( sName := 'a_bPitchExtremeFeatherSoftwareLimitSwitch', sClearName := 'Pitch system detected fine limit', sID := '4090', a := FALSE, b := FALSE, iGroup :=4, iSetDelay :=1, iResetDelay := 10, eResetMode := MANU, eBrakeProgram := B1, eAlarmProgram := 0, Enable := TRUE, iRepetitionNumber := 0 , iRepetitionPeriod := 10, Comment := 'Pitch system detected extreme feather limit', Param1 := (Set:=90, SetMin:=88, SetMax:=90,Comment:=''), Param2 := (Set:=87, SetMin:=87, SetMax:=88,Comment:='') ),
( sName := 'a_bPitchEncoder1Fault', sClearName := 'Pitch system Blade encoder 1', sID := '4091', a := FALSE, b := FALSE, iGroup :=4, iSetDelay :=1, iResetDelay := 1, eResetMode := MANU, eBrakeProgram := B20, eAlarmProgram := 0, Enable := TRUE, iRepetitionNumber := 0 , iRepetitionPeriod := 0, Comment := 'Pitch system Blade encoder 1', Param1 := (Set:=70, SetMin:=28, SetMax:=80,Comment:='Pitch Max motor current exceeded'), Param2 := (Set:=19, SetMin:=0, SetMax:=20,Comment:='') ),
( sName := 'a_bPitchLoadedEFCTest', sClearName := 'Pitch system loaded EFC Test', sID := '4092', a := FALSE, b := FALSE, iGroup :=4, iSetDelay :=1, iResetDelay := 100, eResetMode := MANU, eBrakeProgram := B99, eAlarmProgram := 0, Enable := TRUE, iRepetitionNumber := 0 , iRepetitionPeriod := 0, Comment := 'Pitch system loaded EFC Test', Param1 := (Set:=0, SetMin:=0, SetMax:=0,Comment:=''), Param2 := (Set:=0, SetMin:=0, SetMax:=0,Comment:='') ),
( sName := 'a_bYawDummyAlarm', sClearName := 'Water level below slip ring tripped low sensor', sID := '5001', a := FALSE, b := FALSE, iGroup :=5, iSetDelay :=50, iResetDelay := 0, eResetMode := MANU, eBrakeProgram := B99, eAlarmProgram := 0, Enable := FALSE, iRepetitionNumber := 0 , iRepetitionPeriod := 0, Comment := 'Water level below slip ring tripped low sensor at bottom of trough', Param1 := (Set:=0, SetMin:=0, SetMax:=0,Comment:=''), Param2 := (Set:=0, SetMin:=0, SetMax:=0,Comment:='') ),
( sName := 'a_bLSSDummyAlarm', sClearName := '', sID := '6002', a := FALSE, b := FALSE, iGroup :=5, iSetDelay :=50, iResetDelay := 0, eResetMode := MANU, eBrakeProgram := B100, eAlarmProgram := EMAIL, Enable := FALSE, iRepetitionNumber := 0 , iRepetitionPeriod := 0, Comment := 'Ambient temperature high at front of nacelle', Param1 := (Set:=40, SetMin:=0, SetMax:=100,Comment:=''), Param2 := (Set:=0, SetMin:=0, SetMax:=0,Comment:='') ),
( sName := 'a_bGENDummyAlarm', sClearName := '', sID := '15001', a := FALSE, b := FALSE, iGroup :=5, iSetDelay :=50, iResetDelay := 0, eResetMode := MANU, eBrakeProgram := B100, eAlarmProgram := EMAIL, Enable := FALSE, iRepetitionNumber := 0 , iRepetitionPeriod := 0, Comment := 'Ambient temperature high at front of nacelle', Param1 := (Set:=40, SetMin:=0, SetMax:=100,Comment:=''), Param2 := (Set:=0, SetMin:=0, SetMax:=0,Comment:='') ),
( sName := 'a_bGearDummyAlarm', sClearName := '', sID := '8001', a := FALSE, b := FALSE, iGroup :=5, iSetDelay :=50, iResetDelay := 0, eResetMode := MANU, eBrakeProgram := B100, eAlarmProgram := EMAIL, Enable := FALSE, iRepetitionNumber := 0 , iRepetitionPeriod := 0, Comment := 'Ambient temperature high at front of nacelle', Param1 := (Set:=40, SetMin:=0, SetMax:=100,Comment:=''), Param2 := (Set:=0, SetMin:=0, SetMax:=0,Comment:='') ),
( sName := 'a_bAuxPowerBreakerError_2S1_MainSwitch', sClearName := '2S1', sID := '9001', a := FALSE, b := FALSE, iGroup :=9, iSetDelay :=0, iResetDelay := 0, eResetMode := MANU, eBrakeProgram := B99, eAlarmProgram := 0, Enable := TRUE, iRepetitionNumber := 0 , iRepetitionPeriod := 10, Comment := 'Main Supply Switch', Param1 := (Set:=0, SetMin:=0, SetMax:=0,Comment:=''), Param2 := (Set:=0, SetMin:=0, SetMax:=0,Comment:='') ),
( sName := 'a_bAuxPowerDCbusSupply01Fault', sClearName := 'a_bAuxPowerPriDCbusSupply01Fault', sID := '9038', a := FALSE, b := FALSE, iGroup :=9, iSetDelay :=30, iResetDelay := 0, eResetMode := MANU, eBrakeProgram := B99, eAlarmProgram := 0, Enable := TRUE, iRepetitionNumber := 0 , iRepetitionPeriod := 10, Comment := '', Param1 := (Set:=0, SetMin:=0, SetMax:=0,Comment:=''), Param2 := (Set:=0, SetMin:=0, SetMax:=0,Comment:='') ),
( sName := 'a_bAuxPowerDCbusUPS1AlarmActive', sClearName := 'a_bAuxPowerPriDCbusUPS1AlarmActive', sID := '9039', a := FALSE, b := FALSE, iGroup :=9, iSetDelay :=0, iResetDelay := 0, eResetMode := MANU, eBrakeProgram := B99, eAlarmProgram := 0, Enable := TRUE, iRepetitionNumber := 0 , iRepetitionPeriod := 10, Comment := '', Param1 := (Set:=0, SetMin:=0, SetMax:=0,Comment:=''), Param2 := (Set:=0, SetMin:=0, SetMax:=0,Comment:='') ),
( sName := 'a_bAuxPowerDCbusUPS1BatteryLow', sClearName := 'a_bAuxPowerPriDCbusUPS1BatteryLow', sID := '9040', a := FALSE, b := FALSE, iGroup :=9, iSetDelay :=30, iResetDelay := 0, eResetMode := MANU, eBrakeProgram := B99, eAlarmProgram := 0, Enable := TRUE, iRepetitionNumber := 0 , iRepetitionPeriod := 10, Comment := '', Param1 := (Set:=0, SetMin:=0, SetMax:=0,Comment:=''), Param2 := (Set:=0, SetMin:=0, SetMax:=0,Comment:='') ),
( sName := 'a_bAuxPowerDCbusUPS1BatteryLifeWarning', sClearName := 'a_bAuxPowerPriDCbusUPS1BatteryLifeWarning', sID := '9041', a := FALSE, b := FALSE, iGroup :=9, iSetDelay :=0, iResetDelay := 0, eResetMode := MANU, eBrakeProgram := B99, eAlarmProgram := 0, Enable := TRUE, iRepetitionNumber := 0 , iRepetitionPeriod := 10, Comment := '', Param1 := (Set:=0, SetMin:=0, SetMax:=0,Comment:=''), Param2 := (Set:=0, SetMin:=0, SetMax:=0,Comment:='') ),
( sName := 'a_bAuxPowerDCbusUPS1BatteryLifeLoLo', sClearName := 'a_bAuxPowerPriDCbusUPS1BatteryLifeLoLo', sID := '9042', a := FALSE, b := FALSE, iGroup :=9, iSetDelay :=0, iResetDelay := 0, eResetMode := MANU, eBrakeProgram := B99, eAlarmProgram := 0, Enable := TRUE, iRepetitionNumber := 0 , iRepetitionPeriod := 10, Comment := '', Param1 := (Set:=0, SetMin:=0, SetMax:=0,Comment:=''), Param2 := (Set:=0, SetMin:=0, SetMax:=0,Comment:='') ),
( sName := 'a_bAuxPowerDCbusUPS1BatteryCharging', sClearName := 'a_bAuxPowerPriDCbusUPS1BatteryCharging', sID := '9043', a := FALSE, b := FALSE, iGroup :=9, iSetDelay :=100, iResetDelay := 0, eResetMode := MANU, eBrakeProgram := B99, eAlarmProgram := 0, Enable := TRUE, iRepetitionNumber := 0 , iRepetitionPeriod := 10, Comment := '', Param1 := (Set:=0, SetMin:=0, SetMax:=0,Comment:=''), Param2 := (Set:=0, SetMin:=0, SetMax:=0,Comment:='') ),
( sName := 'a_bAuxPowerDCbusUPS1BatteryChargingTooLong', sClearName := 'a_bAuxPowerPriDCbusUPS1BatteryChargingTooLong', sID := '9044', a := FALSE, b := FALSE, iGroup :=9, iSetDelay :=108000, iResetDelay := 0, eResetMode := MANU, eBrakeProgram := B99, eAlarmProgram := 0, Enable := TRUE, iRepetitionNumber := 0 , iRepetitionPeriod := 10, Comment := '', Param1 := (Set:=0, SetMin:=0, SetMax:=0,Comment:=''), Param2 := (Set:=0, SetMin:=0, SetMax:=0,Comment:='') ),
( sName := 'a_bAuxPowerDCbusORing01RedunFault', sClearName := 'a_bAuxPowerPriDCbusORing01RedunFault', sID := '9045', a := FALSE, b := FALSE, iGroup :=9, iSetDelay :=0, iResetDelay := 0, eResetMode := MANU, eBrakeProgram := B99, eAlarmProgram := 0, Enable := TRUE, iRepetitionNumber := 0 , iRepetitionPeriod := 10, Comment := '', Param1 := (Set:=0, SetMin:=0, SetMax:=0,Comment:=''), Param2 := (Set:=0, SetMin:=0, SetMax:=0,Comment:='') ),
( sName := 'a_bAuxPowerDCbusORing01RedunWarning', sClearName := 'a_bAuxPowerPriDCbusORing01RedunWarning', sID := '9046', a := FALSE, b := FALSE, iGroup :=9, iSetDelay :=0, iResetDelay := 0, eResetMode := MANU, eBrakeProgram := B99, eAlarmProgram := 0, Enable := TRUE, iRepetitionNumber := 0 , iRepetitionPeriod := 10, Comment := '', Param1 := (Set:=0, SetMin:=0, SetMax:=0,Comment:=''), Param2 := (Set:=0, SetMin:=0, SetMax:=0,Comment:='') ),
( sName := 'a_bAuxPowerDCbusDCVoltageLow', sClearName := '', sID := '9074', a := FALSE, b := FALSE, iGroup :=9, iSetDelay :=0, iResetDelay := 0, eResetMode := MANU, eBrakeProgram := B99, eAlarmProgram := 0, Enable := TRUE, iRepetitionNumber := 0 , iRepetitionPeriod := 10, Comment := '24VDC Bus Low Voltage Detected', Param1 := (Set:=23, SetMin:=22, SetMax:=30,Comment:='DC Bus Voltage Low'), Param2 := (Set:=0, SetMin:=0, SetMax:=0,Comment:='') ),
( sName := 'a_bStatusBackupChargerAxis1CriticalError', sClearName := 'a_bStatusBackupChargerAxis1CriticalError', sID := '9074', a := FALSE, b := FALSE, iGroup :=9, iSetDelay :=0, iResetDelay := 0, eResetMode := MANU, eBrakeProgram := B1, eAlarmProgram := 0, Enable := TRUE, iRepetitionNumber := 0 , iRepetitionPeriod := 10, Comment := 'a_bStatusBackupChargerAxis1CriticalError', Param1 := (Set:=0, SetMin:=0, SetMax:=0,Comment:=''), Param2 := (Set:=0, SetMin:=0, SetMax:=0,Comment:='') ),
( sName := 'a_bGridLossDetected', sClearName := '', sID := '10001', a := FALSE, b := FALSE, iGroup :=10, iSetDelay :=0, iResetDelay := 0, eResetMode := MANU, eBrakeProgram := B17, eAlarmProgram := 0, Enable := TRUE, iRepetitionNumber := 0 , iRepetitionPeriod := 10, Comment := 'Grid loss detected by converter', Param1 := (Set:=0, SetMin:=0, SetMax:=0,Comment:=''), Param2 := (Set:=0, SetMin:=0, SetMax:=0,Comment:='') ),
( sName := 'a_bLowVoltageRideThrough', sClearName := '', sID := '10002', a := FALSE, b := FALSE, iGroup :=10, iSetDelay :=0, iResetDelay := 0, eResetMode := MANU, eBrakeProgram := B99, eAlarmProgram := 0, Enable := TRUE, iRepetitionNumber := 0 , iRepetitionPeriod := 10, Comment := 'LVRT detected by converter', Param1 := (Set:=0, SetMin:=0, SetMax:=0,Comment:=''), Param2 := (Set:=0, SetMin:=0, SetMax:=0,Comment:='') ),
( sName := 'a_bScadaEnableAutoStartRequested', sClearName := '', sID := '11001', a := FALSE, b := FALSE, iGroup :=11, iSetDelay :=0, iResetDelay := 0, eResetMode := MANU, eBrakeProgram := B99, eAlarmProgram := 0, Enable := TRUE, iRepetitionNumber := 0 , iRepetitionPeriod := 0, Comment := 'SCADA enable autostart requested', Param1 := (Set:=0, SetMin:=0, SetMax:=0,Comment:=''), Param2 := (Set:=0, SetMin:=0, SetMax:=0,Comment:='') ),
( sName := 'a_bScadaDisableAutoStartRequested', sClearName := '', sID := '11002', a := FALSE, b := FALSE, iGroup :=11, iSetDelay :=0, iResetDelay := 0, eResetMode := MANU, eBrakeProgram := B99, eAlarmProgram := 0, Enable := TRUE, iRepetitionNumber := 0 , iRepetitionPeriod := 0, Comment := 'SCADA disable autostart requested', Param1 := (Set:=0, SetMin:=0, SetMax:=0,Comment:=''), Param2 := (Set:=0, SetMin:=0, SetMax:=0,Comment:='') ),
( sName := 'a_bScadaNormalStopRequested', sClearName := '', sID := '11003', a := FALSE, b := FALSE, iGroup :=11, iSetDelay :=0, iResetDelay := 0, eResetMode := MANU, eBrakeProgram := B99, eAlarmProgram := 0, Enable := TRUE, iRepetitionNumber := 0 , iRepetitionPeriod := 0, Comment := 'SCADA normal stop requested', Param1 := (Set:=0, SetMin:=0, SetMax:=0,Comment:=''), Param2 := (Set:=0, SetMin:=0, SetMax:=0,Comment:='') ),
( sName := 'a_bScadaAlarmResetRequested', sClearName := '', sID := '11004', a := FALSE, b := FALSE, iGroup :=11, iSetDelay :=0, iResetDelay := 0, eResetMode := MANU, eBrakeProgram := B99, eAlarmProgram := 0, Enable := TRUE, iRepetitionNumber := 0 , iRepetitionPeriod := 0, Comment := 'SCADA alarm reset requested', Param1 := (Set:=0, SetMin:=0, SetMax:=0,Comment:=''), Param2 := (Set:=0, SetMin:=0, SetMax:=0,Comment:='') ),
( sName := 'a_bScadaSafetyResetRequested', sClearName := '', sID := '11005', a := FALSE, b := FALSE, iGroup :=11, iSetDelay :=0, iResetDelay := 0, eResetMode := MANU, eBrakeProgram := B99, eAlarmProgram := 0, Enable := TRUE, iRepetitionNumber := 0 , iRepetitionPeriod := 0, Comment := 'SCADA safety reset requested', Param1 := (Set:=0, SetMin:=0, SetMax:=0,Comment:=''), Param2 := (Set:=0, SetMin:=0, SetMax:=0,Comment:='') ),
( sName := 'a_bScadaOpModeChangeRequested', sClearName := '', sID := '11006', a := FALSE, b := FALSE, iGroup :=11, iSetDelay :=0, iResetDelay := 0, eResetMode := MANU, eBrakeProgram := B99, eAlarmProgram := 0, Enable := TRUE, iRepetitionNumber := 0 , iRepetitionPeriod := 0, Comment := 'SCADA op mode change requested', Param1 := (Set:=0, SetMin:=0, SetMax:=0,Comment:=''), Param2 := (Set:=0, SetMin:=0, SetMax:=0,Comment:='') ),
( sName := 'a_bScadaServiceIdleStRequest', sClearName := '', sID := '11007', a := FALSE, b := FALSE, iGroup :=11, iSetDelay :=0, iResetDelay := 0, eResetMode := MANU, eBrakeProgram := B99, eAlarmProgram := 0, Enable := TRUE, iRepetitionNumber := 0 , iRepetitionPeriod := 0, Comment := 'SCADA service idle ST request', Param1 := (Set:=0, SetMin:=0, SetMax:=0,Comment:=''), Param2 := (Set:=0, SetMin:=0, SetMax:=0,Comment:='') ),
( sName := 'a_bScadaServiceStopStRequest', sClearName := '', sID := '11008', a := FALSE, b := FALSE, iGroup :=11, iSetDelay :=0, iResetDelay := 0, eResetMode := MANU, eBrakeProgram := B99, eAlarmProgram := 0, Enable := TRUE, iRepetitionNumber := 0 , iRepetitionPeriod := 0, Comment := 'SCADA service stop ST request', Param1 := (Set:=0, SetMin:=0, SetMax:=0,Comment:=''), Param2 := (Set:=0, SetMin:=0, SetMax:=0,Comment:='') ),
( sName := 'a_bScadaEnableSafetyNACPRequested', sClearName := '', sID := '11009', a := FALSE, b := FALSE, iGroup :=11, iSetDelay :=0, iResetDelay := 0, eResetMode := MANU, eBrakeProgram := B99, eAlarmProgram := 0, Enable := TRUE, iRepetitionNumber := 0 , iRepetitionPeriod := 0, Comment := 'SCADA enable safety NACP requested', Param1 := (Set:=0, SetMin:=0, SetMax:=0,Comment:=''), Param2 := (Set:=0, SetMin:=0, SetMax:=0,Comment:='') ),
( sName := 'a_bScadaDisableSafetyNACPRequested', sClearName := '', sID := '11010', a := FALSE, b := FALSE, iGroup :=11, iSetDelay :=0, iResetDelay := 0, eResetMode := MANU, eBrakeProgram := B99, eAlarmProgram := 0, Enable := TRUE, iRepetitionNumber := 0 , iRepetitionPeriod := 0, Comment := 'SCADA disable safety NACP requested', Param1 := (Set:=0, SetMin:=0, SetMax:=0,Comment:=''), Param2 := (Set:=0, SetMin:=0, SetMax:=0,Comment:='') ),
( sName := 'a_bScadaEnableSafetyNACSRequested', sClearName := '', sID := '11011', a := FALSE, b := FALSE, iGroup :=11, iSetDelay :=0, iResetDelay := 0, eResetMode := MANU, eBrakeProgram := B99, eAlarmProgram := 0, Enable := TRUE, iRepetitionNumber := 0 , iRepetitionPeriod := 0, Comment := 'SCADA enable safety NACS requested', Param1 := (Set:=0, SetMin:=0, SetMax:=0,Comment:=''), Param2 := (Set:=0, SetMin:=0, SetMax:=0,Comment:='') ),
( sName := 'a_bScadaDisableSafetyNACSRequested', sClearName := '', sID := '11012', a := FALSE, b := FALSE, iGroup :=11, iSetDelay :=0, iResetDelay := 0, eResetMode := MANU, eBrakeProgram := B99, eAlarmProgram := 0, Enable := TRUE, iRepetitionNumber := 0 , iRepetitionPeriod := 0, Comment := 'SCADA disable safety NACS requested', Param1 := (Set:=0, SetMin:=0, SetMax:=0,Comment:=''), Param2 := (Set:=0, SetMin:=0, SetMax:=0,Comment:='') ),
( sName := 'a_bScadaLossOfCommsToTTGC', sClearName := '', sID := '11013', a := FALSE, b := FALSE, iGroup :=11, iSetDelay :=0, iResetDelay := 0, eResetMode := MANU, eBrakeProgram := B99, eAlarmProgram := 0, Enable := TRUE, iRepetitionNumber := 0 , iRepetitionPeriod := 0, Comment := 'SCADA loss of comms to TTGC', Param1 := (Set:=0, SetMin:=0, SetMax:=0,Comment:=''), Param2 := (Set:=0, SetMin:=0, SetMax:=0,Comment:='') )];
iMaxAlarms: INT := 222;
arrAlarmStatus: ARRAY [1..222] OF BOOL;
arrAlarmGroup: ARRAY [1..222] OF INT;
END_VAR

// ---- Alarm System/GVLs/A. Operation/01_General/GlobVar_GeneralLog_Privat.TcGVL
{attribute 'Tc2GvlVarNames'}
VAR_GLOBAL	(*GlobVar_GeneralLog_Privat*)

(*-------------  General  / multiple variables  for Operation  --------------------------------------------------------*)

	Lib_rGeneratorPower: 		REAL;
	Lib_rGeneratorSpeed: 		REAL;
	Lib_rFlowSpeed: 			REAL;
(*	Lib_rPitchAngle: 			REAL;	*)


(*-------------  General Log variables  --------------------------------------------------------------------------------------*)

	(* Turbine Identification (Header for log  files):	*)
	Lib_st_xTurbineIdent : 			ST_xTurbineIdent;

	(* System Time:   ---------------------------------------------*)
	Lib_strucSystemTime: 		TIMESTRUCT;
	Lib_sOffsetUTC:			STRING[20];
	Lib_sLocalTime: 			STRING[24];
	Lib_sTimeZoneInfo:		STRING[20];

	(* Operating System:   --------------------------------------*)
	Lib_OperatingSystemCEDetected: 	BOOL;		(*NSM 231016*)
	g_dtLocalTime :DT;
	g_iLocalTime: UDINT;
	g_fLocalTime: LREAL;

(*-------------   In General need for all Logger  --------------------------------------------------------------------------------*)

	LibDetectNewYear	:	BOOL;
	LibDetectNewMonth	:	BOOL;
	LibDetectNewDay		:	BOOL;
	LibDetectNewHour	:	BOOL;
	LibDetectNew10min	:	BOOL;
	LibDetectNew5min	:	BOOL;
	LibDetectNewMinute	:	BOOL;
	LibDetectNew30sec	:	BOOL;
	LibDetectNewSecond	:	BOOL;
	LibDetectNew100ms	:	BOOL;

(* --------------------------------------------------------------------------------------------------------------------------------------*)

END_VAR

// ---- Alarm System/GVLs/A. Operation/01_General/GlobVar_LibStatuscodeLogger_Privat.TcGVL
{attribute 'Tc2GvlVarNames'}
VAR_GLOBAL CONSTANT	(*GlobVar_LibPowerCurves_Privat*)

	guiKeyAndTextLen					: UINT := 91; 		(*max using length for Statuscode description is [uiKeyAndTextLen - sKeySize, e.g. 001-005-280]*)
	NUMBER_OF_EVENT_DATAS			: UINT := 4; 		(* number of process values  *)
	giGeneralLoggerChannelInUsed			: UINT := 75; 		(* how many  channels  the log file max. can contain*)
(*	giNumberOfStatuscodes				: UINT := 850;		*)

	giCountsOfKeyLetterForStatuscodeFile 	: UINT := 75; 		(* Length of minimize Key-string in the file better reading in the text file *)
	giSizeARRListOfStatuscodesToBeSent: 	USINT:= 50;		(*must be tuned to the number given for the ARRAY*)
	guiStrBufferSize: 						UINT:= 47000;		(*length of buffer for statuscode file writing *) (* header 1100 + row 200 * 218 sign = 44700*)

	giHeaderLineLenght					: UINT := 100;		(*length of each line in the header, not the column description*)
	giHeaderColumnLineLEN				: UINT :=4096; 	(*length of column text in the header *)
	giGeneralLenghtOfName				: UINT := 40; 		(* lenght of the column description name *)

END_VAR
VAR_GLOBAL PERSISTENT
//	gxStatuscode		: 				ARRAY[1..850] OF STRUC_Statuscode;
	arrAllListsOfStatuscodesToBeSent: 	ARRAY [1..3] OF ARR_ListOfStatuscodesToBeSent;	(*List of triggered Statuscodes to be sent*)
END_VAR
VAR_GLOBAL

(*  Statuscode Logger:	*)
	gsSC_PathName						: T_MaxString ;	(* Set the Path name in the init program *)
(*	gsSCunlimited_PathName 				: T_MaxString ;	(* Set the Path name with the actual day in the name *)
	gsSCunlimited_PathNameEmbeddedPC	: T_MaxString		:= '\Hard Disk\WEC_Data\Statuscode\';
	gsSCunlimited_PathNamePC 			: T_MaxString 	:='C:\temp\WEC_Data\Statuscode\'; (*Set general name without extension; .txt*)
*)

(*  General Set Values:	*)
	CheckMemCpy_Min	: UDINT;
	CheckMemCpy_Max	: UDINT;
	iOneEntrySize		: INT;
	iOneEntryLength		: INT;

	fbSCLogger					: FB_StatusCodeLogger;
	gwNewDayForLogger    		: WORD; 			(*For detection if we have a new day*)
	giRingBufferFileOneEntryLength 	: UINT; 			(*Length of one entry in the ring buffer Statuscode file*)
	giRingBufferFileHeaderLEN		: INT; 			(*Length of the whole header = header description + column description*)

//	arLoggedSC	 : 				ARRAY[1..400] OF ST_LoggedEvent_SC;	(* Logged Trigger Event *)(* twice(200) - Normal and Transfer Buffers *)
	gstrRingBufferFileColumnText: 	T_MaxString; 		(*first part of column decription*)



	giPointer1AlarmList1: USINT;
	giPointer2AlarmList1: USINT;
	giPointer3AlarmList1: USINT;
	giPointer4AlarmList1: USINT;
	giPointer5AlarmList1: USINT;
	giPointer6AlarmList1: USINT;
	giPointer7AlarmList1: USINT;
	giPointer8AlarmList1: USINT;
	giPointer9AlarmList1: USINT;
	giPointer10AlarmList1: USINT;

	giPointer1AlarmList2: USINT;
	giPointer2AlarmList2: USINT;
	giPointer3AlarmList2: USINT;
	giPointer4AlarmList2: USINT;
	giPointer5AlarmList2: USINT;
	giPointer6AlarmList2: USINT;
	giPointer7AlarmList2: USINT;
	giPointer8AlarmList2: USINT;
	giPointer9AlarmList2: USINT;
	giPointer10AlarmList2: USINT;

	giPointer1AlarmList3: USINT;
	giPointer2AlarmList3: USINT;
	giPointer3AlarmList3: USINT;
	giPointer4AlarmList3: USINT;
	giPointer5AlarmList3: USINT;
	giPointer6AlarmList3: USINT;
	giPointer7AlarmList3: USINT;
	giPointer8AlarmList3: USINT;
	giPointer9AlarmList3: USINT;
	giPointer10AlarmList3: USINT;

	giPointer_fbSendAlarmBuffer1:		USINT;		(*TO_BE_DONE__HP*)	(*pointer must be managed ?????*)
	giPointer_fbSendAlarmBuffer2:		USINT;								(*pointer must be managed ? ? ? ? ?*)
	giPointer_fbSendAlarmBuffer3:		USINT;								(*pointer must be managed ? ? ? ? ?*)


END_VAR

// ---- Alarm System/GVLs/A. Operation/01_General/GVL_Static.TcGVL
{attribute 'Tc2GvlVarNames'}
VAR_GLOBAL
	g_btempAlarmTrig:BOOL;
END_VAR

// ---- Alarm System/GVLs/A. Operation/01_General/ProgramVersions.TcGVL
{attribute 'Tc2GvlVarNames'}
VAR_GLOBAL PERSISTENT

	arrProgramVersions: ARRAY [1..20] OF ST_ProgramVersions :=[
(sVersionDate := '2021_04_21', sChangesMade := '')];
	iMaxProgVersions: INT := 20;
END_VAR

// ---- Alarm System/GVLs/A. Operation/01_General/TurbineData.TcGVL
{attribute 'Tc2GvlVarNames'}
(*VAR_GLOBAL PERSISTENT
 {attribute 'OPC.UA.DA' := '1'}
	stTurbineData: ST_TurbineData :=
	(sOperAlarmParkName :='',
	sOperAlarmTurbineName :='',
	sOperAlarmParkId :='',
	sOperAlarmTurbineId :='',
	sOperCountryCode :='',
	sOperTurbineManufacturer :='',
	sOperTurbineType :='',
	sOperBladeType := '',
	sOperInverterType := '',
	sOperTowerType := '',
	sOperTowerBearing := '',
	sTower1stBendFreg := '',
	sTower2ndBendFreg := '',
	sPitchGenNomSpeed := '');		

END_VAR
*)

VAR_GLOBAL
//	g_stTurbineRelatedData: ST_TurbineRelatedData;
 {attribute 'OPC.UA.DA' := '1'}
	g_bOperTurbineCommsFault: BOOL;
	 {attribute 'OPC.UA.DA' := '1'}
	g_fOperTurbineCapacityFactor :REAL;
   {attribute 'OPC.UA.DA' := '1'}
	g_fOperTurbineTotalEnergyGenerated :REAL;
   {attribute 'OPC.UA.DA' := '1'}
	g_tOperTurbineTimeSpentInFaultState :TIME;
   {attribute 'OPC.UA.DA' := '1'}
	g_tOperTurbineTimeSpentInOffState :TIME;
   {attribute 'OPC.UA.DA' := '1'}
	g_tOperTurbineTimeSpentInProduction :TIME;  

END_VAR

// ---- Alarm System/GVLs/GVL_EventLogger.TcGVL
{attribute 'qualified_only'}
VAR_GLOBAL
	cMaxNumberOfEvent:UINT; //
	
	
	
END_VAR

// ---- Base/Example/GVL/GVL_HMI.TcGVL
{attribute 'qualified_only'}
VAR_GLOBAL
	(*IO*)
	stTest04_DigitalInput:stHMI_DigitalInput;
	stTest05_DigitalInput:stHMI_DigitalInput;
	
	(*SYSTEM*)
	stTest01_Intlk:stHMI_Interlock;
	stTest02_Perm:stHMI_Permissive;
	stTest03_RunCtrl:stHMI_SystemRunControl;
END_VAR

// ---- MAIN.TcPOU
PROGRAM MAIN
VAR
	
END_VAR

POU_TestBase();

//AlarmWithCustomSourceInfo();
//OtherAlarmsWithCustomSource();
P_AlarmHandling();
P_AlarmTable();
MultipleAlarmCreation();

P_EventLogger_TCSAlarms();

END_PROGRAM

// ---- Base/Example/POU/POU_TestBase.TcPOU
PROGRAM POU_TestBase
VAR
	fbTestAI:fbIO_AnalogueInput;
	fbTestIntlk:FB_Interlock;	
	fbTestPerm:FB_Permissive;
	fbTestRunCtrl:FB_SystemRunControl;
	fbTestDigitalInput:fbIO_DigitalInput;
	HMI_AI_001:stHMI_AnalogueInput;
	ERROR_AI_001:stError_AnalogueInput;
	fbTestAO:fbIO_AnalogueOutput;
	HMI_DI_001:stHMI_DigitalInput;
	pulseTest:fbPulser;
	HMI_DO_001:stHMI_DigitalOutput;
	fbTestDO:fbIO_DigitalOutput;
	testAlarmset:FB_AlarmEventSet;
	bHMITest:BOOL;
	bPLCTest:BOOL;
	
	test_Valve:fbValve_Solenoid;
	HMI_XV_001:stHMI_ValveControl;
	Error_XV_001:stError_Valve;
END_VAR

testAlarmset(bAlarmEventTrigger:= , tSetDelay:= , tResetDelay:= , bOutAlarmEvent=> );

test_Valve(
	tInTimeout:= , 
	iInMode:= , 
	bInEstop:= , 
	bInSignalHome:= , 
	bInSignalWork:= , 
	bInEnable:= , 
	bInCommandWork:= , 
	bInResetError:= , 
	bInSimulate:= , 
	bOutCommandHome=> , 
	bOutCommandWork=> , 
	bOutActiveHome=> , 
	bOutActiveWork=> , 
	bOutAuto=> , 
	bOutError=> , 
	ERROR_Valve=>Error_XV_001 , 
	HMI_ValveControl:=HMI_XV_001 );

fbTestDigitalInput(
	iInMode:= , 
	bInInput:= , 
	tInOnDebounce:= , 
	tInOffDebounce:= , 
	bOutAuto=> , 
	bOutOn=> , 
	bOutRisingEdge=> , 
	bOutFallingEdge=> , 
	HMI_DigitalInput:=HMI_DI_001 );

fbTestAI(
	iInMode:= , 
	iInValue:= , 
	iInSensorType:= , 
	rInEngUnitsMin:= , 
	rInEngUnitsMax:= , 
	rInLowLow:= , 
	rInLow:= , 
	rInHigh:= , 
	rInHighHigh:= , 
	rInLowLowDeadband:= , 
	rInLowDeadband:= , 
	rInHighDeadband:= , 
	rInHighHighDeadband:= , 
	bInResetError:= , 
	rOutEngUnitsValue=> , 
	bOutLowLow=> , 
	bOutLow=> , 
	bOutHigh=> , 
	bOutHighHigh=> , 
	bOutAuto=> , 
	bOutError=> , 
	ERROR_IO_AnalogueIn=>ERROR_AI_001 , 
	HMI_IO_AnalogueInput:=HMI_AI_001 );
	
fbTestIntlk(
	bInterlock1:= , 
	bInterlock2:= , 
	bInterlock3:= , 
	bInterlock4:= , 
	bInterlock5:= , 
	bInterlock6:= , 
	bInterlock7:= , 
	bInterlock8:= , 
	bInterlock9:= , 
	bInterlock10:= , 
	bInterlock11:= , 
	bInterlock12:= , 
	bInterlock13:= , 
	bInterlock14:= , 
	bInterlock15:= , 
	bInterlock16:= , 
	bOutInterlockOk=> , 
	HMI_Interlock:=GVL_HMI.stTest01_Intlk );

fbTestPerm(
	bPermissive1:= , 
	bPermissive2:= , 
	bPermissive3:= , 
	bPermissive4:= , 
	bPermissive5:= , 
	bPermissive6:= , 
	bPermissive7:= , 
	bPermissive8:= , 
	bPermissive9:= , 
	bPermissive10:= , 
	bPermissive11:= , 
	bPermissive12:= , 
	bPermissive13:= , 
	bPermissive14:= , 
	bPermissive15:= , 
	bPermissive16:= , 
	bOutPermissiveOk=>, 
	HMI_Permissive:= GVL_HMI.stTest02_Perm);

GVL_HMI.stTest01_Intlk.asInterlockNames[1]:='Valve in correct pos';
	
fbTestRunCtrl(
	bInEnableStart:= , 
	bInEnableStop:= , 
	bInStartAuto:= , 
	bInStopAuto:= , 
	bOutRunCmd=> , 
	HMI_SystemRunControl:= GVL_HMI.stTest03_RunCtrl);
	
fbTestDO(
	iInMode:= , 
	bInEstop:= , 
	bInEnable:= , 
	bInCommand:= , 
	bOutAuto=> , 
	bOutCommand=> , 
	HMI_IO_DigitalOutput:=HMI_DO_001 );

pulseTest(
	bInRun:= , 
	tInTimeOn:=T#5S , 
	tInTimeOff:=T#10S , 
	iInNumPulses:= , 
	bOutPulse=> , 
	bOutDone=> , 
	iOutCount=> );
	
	POu();

END_PROGRAM

// ---- Base/IO/POU/fbIO_AnalogueInput.TcPOU
FUNCTION_BLOCK fbIO_AnalogueInput
VAR_INPUT
	iInMode:		INT;
	iInValue:		INT;
	iInSensorType:	INT;
	rInEngUnitsMin:	REAL;
	rInEngUnitsMax:	REAL;
	rInLowLow:		REAL;
	rInLow:			REAL;
	rInHigh:		REAL;
	rInHighHigh:	REAL;
	rInLowLowDeadband: REAL;
	rInLowDeadband:REAL;
	rInHighDeadband:REAL;
	rInHighHighDeadband:REAL;
	bInResetError:BOOL;
END_VAR
VAR_OUTPUT
	rOutEngUnitsValue:REAL; (*Engineering units scaled value*)
	bOutLowLow:BOOL; (*Low low alarm is active*)
	bOutLow:BOOL; (*Low warning is active*)
	bOutHigh:BOOL; (*High warning is active*)
	bOutHighHigh:BOOL; (*High high alarm is active*)
	bOutAuto:BOOL; (*Input is in auto mode*)
	bOutError:BOOL; (*Error Exists*)
	ERROR_IO_AnalogueIn:stError_AnalogueInput;
END_VAR

VAR_IN_OUT
	HMI_IO_AnalogueInput:stHMI_AnalogueInput;
END_VAR

VAR
	fScaled16:REAL;
	fTempScaled16:REAL;
	ftempScaled16_a:REAL;
	ftempScaled16_b:REAL;
	bTest:BOOL;
END_VAR

//Process Alarms limits
bOutLowLow:= (rOutEngUnitsValue<=(rInLowLow-rInLowLowDeadband));  	// LL Alarm
bOutLow:= (rOutEngUnitsValue<=(rInLow-rInLowDeadband));  			// LL Warning
bOutHighHigh:= (rOutEngUnitsValue>=(rInHigh+rInHighHighDeadband));  	// HH Alarm	
bOutHigh:= (rOutEngUnitsValue>=(rInHighHigh+rInHighDeadband));  		// HH Warning	
	
bOutAuto := iInMode=1;

(***************************SCALING ANALOGUE************************
ftempScaled16_a:=
ftempScaled16_b:=
IF fTempScaled32 THEN
	
END_IF
*)
(*
CASE iInMode OF
	0:
		;
	1:	// Auto mode
		rOutEngUnitsValue:=fScaled16;
	2:	// Manual Mode
		rOutEngUnitsValue:=HMI_IO_AnalogueInput.rManualValue;
		
	3:	// Independant
	END_CASE
*)

(*control bOut based on the global input and HMI input mode*)
(*if in independant mode allow control of the output based on HMI commands (MANUAL) AND digital input (AUTO)*)
IF iInMode=10 THEN
	//if HMI requests manual mode 
	IF HMI_IO_AnalogueInput.iMode=2 THEN
		;
	ELSE
		;
	END_IF
ELSE
	//bOutOn:=tonInOnDebounce.Q OR tofInOnDebounce.Q;
END_IF
	


(*Map Error bits*)
ERROR_IO_AnalogueIn.LowLowAlarm:=bOutLowLow;			//HH alarm
ERROR_IO_AnalogueIn.HighHighAlarm:=bOutHighHigh;		//LL Alarm	
	
(*map active value to the scada*)
HMI_IO_AnalogueInput.rInputValue:=fScaled16;
HMI_IO_AnalogueInput.rActiveValue:=rOutEngUnitsValue;

(*Error Code*)
HMI_IO_AnalogueInput.iErrorCode.0:=ERROR_IO_AnalogueIn.LowLowAlarm;	
HMI_IO_AnalogueInput.iErrorCode.1:=ERROR_IO_AnalogueIn.HighHighAlarm;	
HMI_IO_AnalogueInput.iErrorCode.2:=ERROR_IO_AnalogueIn.LowLowAlarm;	
HMI_IO_AnalogueInput.iErrorCode.3:=bTest;
	
HMI_IO_AnalogueInput.bError:=(HMI_IO_AnalogueInput.iErrorCode<>0);

END_FUNCTION_BLOCK

// ---- Base/General Control/POU/FB_Interlock.TcPOU
FUNCTION_BLOCK FB_Interlock
VAR_INPUT
	bInterlock1:BOOL;
	bInterlock2:BOOL;
	bInterlock3:BOOL;
	bInterlock4:BOOL;
	bInterlock5:BOOL;
	bInterlock6:BOOL;
	bInterlock7:BOOL;
	bInterlock8:BOOL;
	bInterlock9:BOOL;
	bInterlock10:BOOL;
	bInterlock11:BOOL;
	bInterlock12:BOOL;
	bInterlock13:BOOL;
	bInterlock14:BOOL;
	bInterlock15:BOOL;
	bInterlock16:BOOL;
END_VAR

VAR_OUTPUT
	bOutInterlockOk:BOOL;	(*1=System ok to operate*)
END_VAR

VAR_IN_OUT
	HMI_Interlock:stHMI_Interlock;
END_VAR

VAR
	wInterlock:WORD;
	wInterlockMask:WORD:=16#FFFF;
END_VAR

(*Map interlock status*)
wInterlock.0:=HMI_Interlock.abInterlocks[1]:=bInterlock1;
wInterlock.1:=HMI_Interlock.abInterlocks[2]:=bInterlock2;
wInterlock.2:=HMI_Interlock.abInterlocks[3]:=bInterlock3;
wInterlock.3:=HMI_Interlock.abInterlocks[4]:=bInterlock4;
wInterlock.4:=HMI_Interlock.abInterlocks[5]:=bInterlock5;
wInterlock.5:=HMI_Interlock.abInterlocks[6]:=bInterlock6;
wInterlock.6:=HMI_Interlock.abInterlocks[7]:=bInterlock7;
wInterlock.7:=HMI_Interlock.abInterlocks[8]:=bInterlock8;
wInterlock.8:=HMI_Interlock.abInterlocks[9]:=bInterlock9;
wInterlock.9:=HMI_Interlock.abInterlocks[10]:=bInterlock10;
wInterlock.10:=HMI_Interlock.abInterlocks[11]:=bInterlock11;
wInterlock.11:=HMI_Interlock.abInterlocks[12]:=bInterlock12;
wInterlock.12:=HMI_Interlock.abInterlocks[13]:=bInterlock13;
wInterlock.13:=HMI_Interlock.abInterlocks[14]:=bInterlock14;
wInterlock.14:=HMI_Interlock.abInterlocks[15]:=bInterlock15;
wInterlock.15:=HMI_Interlock.abInterlocks[16]:=bInterlock16;

(*check active interlocks with the interlock mask set interlock ok status*)
IF (wInterlock AND wInterlockMask)=wInterlockMask THEN
	bOutInterlockOk:=1;
END_IF

END_FUNCTION_BLOCK

// ---- Base/General Control/POU/FB_Permissive.TcPOU
FUNCTION_BLOCK FB_Permissive
VAR_INPUT
	bPermissive1:BOOL;
	bPermissive2:BOOL;
	bPermissive3:BOOL;
	bPermissive4:BOOL;
	bPermissive5:BOOL;
	bPermissive6:BOOL;
	bPermissive7:BOOL;
	bPermissive8:BOOL;
	bPermissive9:BOOL;
	bPermissive10:BOOL;
	bPermissive11:BOOL;
	bPermissive12:BOOL;
	bPermissive13:BOOL;
	bPermissive14:BOOL;
	bPermissive15:BOOL;
	bPermissive16:BOOL;
END_VAR

VAR_OUTPUT
	bOutPermissiveOk:BOOL;	(*1=System ok to operate*)
END_VAR

VAR_IN_OUT
	HMI_Permissive:stHMI_Permissive;
END_VAR

VAR
	wPermissive:WORD;
	wPermissiveMask:WORD:=16#FFFF;
END_VAR

wPermissive.0:=HMI_Permissive.abPermissives[1]:=bPermissive1;
wPermissive.1:=HMI_Permissive.abPermissives[2]:=bPermissive2;
wPermissive.2:=HMI_Permissive.abPermissives[3]:=bPermissive3;
wPermissive.3:=HMI_Permissive.abPermissives[4]:=bPermissive4;
wPermissive.4:=HMI_Permissive.abPermissives[5]:=bPermissive5;
wPermissive.5:=HMI_Permissive.abPermissives[6]:=bPermissive6;
wPermissive.6:=HMI_Permissive.abPermissives[7]:=bPermissive7;
wPermissive.7:=HMI_Permissive.abPermissives[8]:=bPermissive8;
wPermissive.8:=HMI_Permissive.abPermissives[9]:=bPermissive9;
wPermissive.9:=HMI_Permissive.abPermissives[10]:=bPermissive10;
wPermissive.10:=HMI_Permissive.abPermissives[11]:=bPermissive11;
wPermissive.11:=HMI_Permissive.abPermissives[12]:=bPermissive12;
wPermissive.12:=HMI_Permissive.abPermissives[13]:=bPermissive13;
wPermissive.13:=HMI_Permissive.abPermissives[14]:=bPermissive14;
wPermissive.14:=HMI_Permissive.abPermissives[15]:=bPermissive15;
wPermissive.15:=HMI_Permissive.abPermissives[16]:=bPermissive16;

IF (wPermissive AND wPermissiveMask)=wPermissiveMask THEN
	bOutPermissiveOk:=1;
END_IF

END_FUNCTION_BLOCK

// ---- Base/General Control/POU/FB_SystemRunControl.TcPOU
FUNCTION_BLOCK FB_SystemRunControl
VAR_INPUT
	bInEnableStart:BOOL; (*Interlocks the system from being able to start running*)
	bInEnableStop:BOOL; (*Interlocks the system FROM being able TO stop*)
	bInStartAuto:BOOL;	(*Starts the system running in auto mode*)
	bInStopAuto:BOOL;	(*Stop the system in auto mode*)
END_VAR
VAR_OUTPUT
	bOutRunCmd:BOOL;
END_VAR

VAR_IN_OUT
	HMI_SystemRunControl:stHMI_SystemRunControl;
END_VAR

VAR
	bStart:BOOL;
	bStop:BOOL;
END_VAR

bStart := (bInEnableStart) AND (bInStartAuto OR (HMI_SystemRunControl.bPBEN_Start AND HMI_SystemRunControl.bPB_Start));
bStop  := (bInEnableStop) AND (bInStopAuto OR (HMI_SystemRunControl.bPBEN_Stop AND HMI_SystemRunControl.bPBEN_Stop));

bOutRunCmd := HMI_SystemRunControl.bRunning := bStart AND NOT(bStop);

END_FUNCTION_BLOCK

// ---- Base/IO/POU/fbIO_DigitalInput.TcPOU
FUNCTION_BLOCK fbIO_DigitalInput
VAR_INPUT
	iInMode:INT;				(*global mode input 0=stop, 1=Auto, 2=Manuall,10=Independant*)
	bInInput:BOOL; 				(*The raw digital input signal*)
	tInOnDebounce:TIME:=T#0MS;	(*Optional debounce timer for rising edge of input (T#0ms to disable)*)
	tInOffDebounce:TIME:=T#0MS;	(*Optional debounce timer for falling edge of input (T#0ms to disable)*)
END_VAR
VAR_OUTPUT
	bOutAuto:BOOL;		  (* Block in auto mode*)
	bOutOn:BOOL;		  (*The status of the digital input*)
	bOutRisingEdge:BOOL;  (*The status of the input transitioned FROM low TO high. TRUE FOR exactly 1 scan*)
	bOutFallingEdge:BOOL; (*The status of the input transitioned FROM high TO low. TRUE FOR exactly 1 scan*)
END_VAR

VAR_IN_OUT
	HMI_DigitalInput:stHMI_DigitalInput;
END_VAR

VAR
	tonInOnDebounce:TON;
	tofInOnDebounce:TOF;
	rTrigbInput:R_TRIG;
	fTrigbInput:F_TRIG;
END_VAR

(*debounce logic - output read after debounce  time*)
tonInOnDebounce(IN:=bInInput, PT:=tInOnDebounce, );
tofInOnDebounce(IN:=bInInput , PT:=tInOffDebounce );

(*map edge triggered outputs*)
rTrigbInput(CLK:=bInInput , Q=>bOutRisingEdge );
fTrigbInput(CLK:=bInInput , Q=>bOutFallingEdge );

(*control bOut based on the global input and HMI input mode*)
(*if in independant mode allow control of the output based on HMI commands (MANUAL) AND digital input (AUTO)*)
IF iInMode=10 THEN
	//if HMI requests manual mode 
	IF HMI_DigitalInput.iMode=2 THEN
		IF HMI_DigitalInput.bPBEN_On AND HMI_DigitalInput.bPB_On THEN
			bOutOn:=1;
		ELSIF HMI_DigitalInput.bPBEN_Off AND HMI_DigitalInput.bPB_Off THEN
			bOutOn:=0;
		END_IF
	ELSE
		bOutOn:=tonInOnDebounce.Q OR tofInOnDebounce.Q;   /// auto output
	END_IF
ELSE
	bOutOn:=tonInOnDebounce.Q OR tofInOnDebounce.Q;
END_IF

(*map auto status output*)
bOutAuto:=(iInMode<>2) AND (HMI_DigitalInput.iMode<>2);

(*map HMI_DigitalInput outputs*)
HMI_DigitalInput.bOnActual:=tofInOnDebounce.Q OR tonInOnDebounce.Q;
HMI_DigitalInput.bOn:=bOutOn;

END_FUNCTION_BLOCK

// ---- Base/IO/POU/fbIO_AnalogueOutput.TcPOU
FUNCTION_BLOCK fbIO_AnalogueOutput
VAR_INPUT
	iInMode: INT; //Mode input
	iInSensorType :INT;		//Enumerated value of of sensor types
	iInEstopFunction: INT; 	(*maximum set point (rInEngUnitsMin), and ‘Estop.HMISetPoint’ sets to an HMspecified value that can be in between the min and max*)
	bInEstop:BOOL;			//Emergency stop input
	bInEnable:BOOL;			//Interlock for the Analog Output. If this bit is false, then output will be 0
	rInValue:REAL;			//Auto mode value of output
	rInEngUnitsMin	:REAL; 	//Engineering units scale min
	rInEngUnitsMax: REAL;	//Engineering units scale max
	bInResetError: BOOL;	//If an error condition exists, the error must be fixed first, then set this bit high to reset the internal error
END_VAR
VAR_OUTPUT
	bOutAuto:BOOL;									//Block in auto mode		
	bOutError:BOOL;									//Error exists
	wOutValue:WORD;									//Value to output to Analog Output
	ERROR_IO_AnalogueOut: stError_AnalogueOutput;   //This output UDT has one bit for every type of error. It should be mapped to 
													//the HMI’s error list. It can also be used for advanced debugging of the error state*)
END_VAR
VAR_IN_OUT
	HMI_IO_AnalogOutput:stHMI_AnalogueOutput;		//struct used to communicate with the HMI
END_VAR
VAR
END_VAR

(*Map HMI structures elements*)
HMI_IO_AnalogOutput.bInterlock:=bInEnable;
HMI_IO_AnalogOutput.rAutoValue:=rInValue;


CASE iInMode OF
	0:
		;
	1:	// Auto mode
		wOutValue:=0;
	2:	// Manual Mode
		//wOutValue:=HMI_IO_AnalogOutput.rManualValue;
	3:	// Independant
	;
END_CASE

(*Map ERROR_IO_AnalogueOut Structure*)

END_FUNCTION_BLOCK

// ---- Base/Process Control/POU/fbPulser.TcPOU
FUNCTION_BLOCK fbPulser
VAR_INPUT
	bInRun:		BOOL;	(*Enables the pulsing output*)
	tInTimeOn:	TIME;	(*Amount of time output is turned on each period*)
	tInTimeOff:	TIME;	(*Amount of time output is off each period*)
	iInNumPulses: INT;	(*Number of pulses to output (0 for infinite)*)
END_VAR
VAR_OUTPUT
	bOutPulse:	BOOL;	(*The pulsing output*)
	bOutDone:	BOOL;	(*Pulsing complete, iNumPulses achieved*)
	iOutCount:	INT;	(*Current number of pulses complete*)

END_VAR
VAR
	rTrigbRun:R_TRIG;
	nState: INT;
	tonTimerOn:TON;
	tonTimerOff:TON;
END_VAR

rTrigbRun(CLK:=bInRun , Q=> );

//When a new run command is issued the pulsing sequence is restarted
IF rTrigbRun.Q THEN
	nState:=10;
END_IF

CASE nstate OF
	0:
		bOutPulse:=0;
		iOutCount:=0;
		
	10:
		bOutPulse:=1;
		IF NOT(bInRun) OR bOutDone THEN
			nState:=0;
		ELSIF tonTimerOn.Q THEN
			iOutCount:=iOutCount+1;
			nState:=20;
		END_IF	
	20:
		bOutPulse:=0;
		IF NOT(bInRun) OR bOutDone THEN
			nState:=0;
		ELSIF tonTimerOff.Q THEN
			nState:=10;
		END_IF	
		
END_CASE

bOutDone:=(iOutCount>=iInNumPulses) AND NOT(iInNumPulses=0);  // run infinitely if inumpulse=0
tonTimerOn(IN:=(nState=10) , PT:=tInTimeOn , Q=> , ET=> );	  // time in state 10 -- time pulse on	
tonTimerOff(IN:=(nState=20) , PT:=tInTimeOff , Q=> , ET=> );	  // time in state 20 -- time pulse off

END_FUNCTION_BLOCK

// ---- Base/IO/POU/fbIO_DigitalOutput.TcPOU
FUNCTION_BLOCK fbIO_DigitalOutput
VAR_INPUT
	iInMode:INT;		(*global mode input*)
	bInEstop:BOOL;		(* Emergency stop input 1=Estop Active*)
	bInEnable:BOOL;		(*Interlock for the digital output. If this bit is false, then output will be 0*)
	bInCommand:BOOL;	(*The command to the digital output*)
END_VAR
VAR_OUTPUT
	bOutAuto:BOOL;		(*Block in auto mode*)
	bOutCommand:BOOL;	(*Command to digital output*)
END_VAR
VAR_IN_OUT
	HMI_IO_DigitalOutput:stHMI_DigitalOutput;
END_VAR
VAR
	bTempOutCommand:BOOL;
	bSetHMICommandsOFF:BOOL;
END_VAR

(*control bOut based on the global input and HMI input mode*)
(*if in independant mode allow control of the output based on HMI commands (MANUAL) AND digital input (AUTO)*)
IF iInMode=10 THEN
	//if HMI requests manual mode 
	IF HMI_IO_DigitalOutput.iMode=2 THEN
		bOutAuto:=0;
		bSetHMICommandsOFF:=0;
		IF HMI_IO_DigitalOutput.bPBEN_On AND HMI_IO_DigitalOutput.bPB_On THEN
			bTempOutCommand:=1;
		ELSIF HMI_IO_DigitalOutput.bPBEN_Off AND HMI_IO_DigitalOutput.bPB_Off THEN
			bTempOutCommand:=0;
		END_IF
	ELSE
		bTempOutCommand:=bInCommand;   /// auto output
		bOutAuto:=1;
		bSetHMICommandsOFF:=1;
	END_IF
ELSE
	bTempOutCommand:=bInCommand;   /// auto output
	bSetHMICommandsOFF:=1;
	bOutAuto:=1;
END_IF

bOutCommand := bTempOutCommand AND  bInEnable AND bInEstop;//allow output when interlocked and Estop ok

HMI_IO_DigitalOutput.bCommandAuto:=bInCommand;
HMI_IO_DigitalOutput.bCommand:=bTempOutCommand;
HMI_IO_DigitalOutput.bInterlock:=bInEnable;

IF bSetHMICommandsOFF THEN
	HMI_IO_DigitalOutput.iMode:=1;
	HMI_IO_DigitalOutput.bPBEN_On:=0;
	HMI_IO_DigitalOutput.bPBEN_Off:=0;
	HMI_IO_DigitalOutput.bPB_On:=0;
	HMI_IO_DigitalOutput.bPB_Off:=0;
END_IF

END_FUNCTION_BLOCK

// ---- Base/General Control/POU/FB_AlarmEventSet.TcPOU
FUNCTION_BLOCK FB_AlarmEventSet
VAR_INPUT
	bAlarmEventTrigger:BOOL;
	tSetDelay:TIME;
	tResetDelay:TIME;
	bManualReset:BOOL;
	bResetError:BOOL;
	bEnableAlarm:BOOL;
END_VAR
VAR_OUTPUT
	bOutAlarmEvent:	BOOL;
END_VAR
VAR
	
	bReset:BOOL;
	TON_SetDelay:TON;
	TON_ResetDelay:TOF;
	Latch:SR;
END_VAR

IF (bManualReset AND bResetError AND NOT(bAlarmEventTrigger))
	OR (NOT(bManualReset) AND NOT(bAlarmEventTrigger))  OR NOT(bEnableAlarm) THEN
	bReset:=1;
ELSE
	bReset:=0;
END_IF

Latch(SET1:=TON_SetDelay.Q , 
	  RESET:=bReset , 
	  Q1=> );

TON_ResetDelay(IN:=Latch.Q1 , PT:=tResetDelay , Q=> , ET=> );
TON_SetDelay(IN:=bAlarmEventTrigger AND bEnableAlarm, PT:=tSetDelay , Q=> , ET=> );

bOutAlarmEvent:=TON_ResetDelay.Q;

END_FUNCTION_BLOCK

// ---- Base/Valve Control/POU/fbValve_Solenoid.TcPOU
FUNCTION_BLOCK fbValve_Solenoid
VAR_INPUT
	tInTimeout: TIME:=T#10S;		//The amount of time before an error condition triggers an error
	iInMode:	INT;		//system mode 1=Auto, 2=Manual, 10=Independent
	bInEstop:	BOOL;		//Emergency stop input 1=Estop
	bInSignalHome:	BOOL;	//Home position feedback
	bInSignalWork:	BOOL;	//Work position feedback
	bInEnable:		BOOL;	//Valve interlock. The valve is allowed to operate if this condition has been met
	bInCommandWork: BOOL;	//Move to work position in automatic mode
	bInResetError:	BOOL;	//If an error condition exists, the error must be fixed first, then set this bit high to reset the internal error
	bInSimulate:	BOOL;	//Enables software simulation of device.
END_VAR
VAR_OUTPUT
	bOutCommandHome: BOOL;	//Output for home position
	bOutCommandWork: BOOL;	//Output for work position
	bOutActiveHome: BOOL;	//Valve is actively in home position
	bOutActiveWork: BOOL;	//Valve is actively in work position
	bOutAuto: BOOL;			//This output indicates whether the block is in auto mode
	bOutError: BOOL;		//This output indicates whether there's an error condition in the cylinder
	ERROR_Valve:stError_Valve;
END_VAR

VAR_IN_OUT
	HMI_ValveControl:stHMI_ValveControl;
END_VAR

VAR
	tonTimeOut:TON;
	iErrorCode:INT;
	bNewMode:BOOL;	 (*new mode selected*)
	bAutoMode:BOOL;	 (*Automode active*)
	bManualMode:BOOL; (*Manual Mode active*)
	iLastMode:INT;	(*last mode code*)
	bEnableHome:BOOL;	 (*home position enabled*)
	bEnableWork:BOOL;	 (*work position enabled*)
	bPB_Home:BOOL;		 (*PB Move to home in manual mode*)
	bPB_Work:BOOL;		 (*PB Move to work in manual mode*)
	bPB_ResetError:BOOL; (*PB Reset error*)
	bReset: BOOL;
END_VAR



(*****************************INPUTS*************************************************)
(*Read HMI input button*)

fcHMIBit(bInToggle:=0 , bInLatch:=0 , bHMI:=HMI_ValveControl.bPB_Home , bPLC:=bPB_Home );
fcHMIBit(bInToggle:=0 , bInLatch:=0 , bHMI:=HMI_ValveControl.bPB_Work , bPLC:=bPB_Work );
fcHMIBit(bInToggle:=0 , bInLatch:=0 , bHMI:=HMI_ValveControl.bPB_ResetError , bPLC:=bPB_ResetError );
(*update the signal home bit*)
HMI_ValveControl.bSignalHome:=bInSignalHome;

(*update the signal work bit*)
HMI_ValveControl.bSignalWork:=bInSignalWork;

(**************************CONTROL LOGIC************************************************)
(*Clear all errors*)
IF (bInResetError OR bPB_ResetError) AND HMI_ValveControl.bPB_ResetError THEN
	bReset:=1;
ELSE 
	bReset:=0;
END_IF


(*override HMI mode if not in Independant mode*)
IF iInMode<>10 THEN
	HMI_ValveControl.iMode:=iInMode;
END_IF

(*detect change in mode*)
bNewMode:=HMI_ValveControl.iMode<>iLastMode;

(*keep track of last mode*)
iLastMode:=HMI_ValveControl.iMode;

(*Determine if auto or manual mode Active*)
bManualMode:=NOT(bInEstop) AND NOT(bNewMode) AND (HMI_ValveControl.iMode=2);
bAutoMode:=NOT(bInEstop) AND NOT(bNewMode) AND (HMI_ValveControl.iMode=1);

(*Enable home and work positions*)
bEnableWork:=bEnableHome:= NOT(HMI_ValveControl.bError) AND (bManualMode OR bAutoMode);

HMI_ValveControl.bPBEN_Home:=HMI_ValveControl.bPBEN_Work:=bManualMode AND NOT(HMI_ValveControl.bError);

(*enable error reset button if error present*)
HMI_ValveControl.bPBEN_ResetError:=HMI_ValveControl.bPB_ResetError;

(*Command Home position*)
IF (bManualMode AND bPB_Home AND  NOT(bPB_Work) AND HMI_ValveControl.bPBEN_Home) OR
	(bAutoMode AND NOT(bInCommandWork) AND bEnableHome) THEN
	HMI_ValveControl.bHomeOn:=1;
	HMI_ValveControl.bWorkOn:=0;
END_IF

(*command work position*)
IF (bManualMode AND bPB_Work AND  NOT(bPB_Home) AND HMI_ValveControl.bPBEN_Work) OR
	(bAutoMode AND bInCommandWork AND bEnableWork) THEN
	HMI_ValveControl.bWorkOn:=1;
	HMI_ValveControl.bHomeOn:=0;
END_IF

(*reset work if not enabled*)
IF bAutoMode AND NOT(bEnableWork) THEN
	HMI_ValveControl.bWorkOn:=0;
END_IF

(*reset home if not enabled*)
IF bAutoMode AND NOT(bEnableHome) THEN
	HMI_ValveControl.bHomeOn:=0;
END_IF

(*if Not in auto or manual reset both*)
IF NOT(bAutoMode OR bManualMode) THEN
	HMI_ValveControl.bHomeOn:=0;
	HMI_ValveControl.bWorkOn:=0;
END_IF

(************************************ERRORS*************************************************************)
(*set timeout errors*)
tonTimeOut(IN:=HMI_ValveControl.bHomeOn OR HMI_ValveControl.bWorkOn , PT:= , Q=> , ET=> );

(*Error: Work Feedback not active*)
ERROR_Valve.NoWorkFeedback:=NOT(bInEstop) AND tonTimeOut.Q AND HMI_ValveControl.bWorkOn AND NOT(HMI_ValveControl.bSignalWork);

(*Error: Home feedback not active*)
ERROR_Valve.NoHomeFeedback:=NOT(bInEstop) AND tonTimeOut.Q AND HMI_ValveControl.bHomeOn AND NOT(HMI_ValveControl.bSignalHome);

(*Error: Home position still active*)
ERROR_Valve.HomeFeedbackStillActive:=NOT(bInEstop) AND tonTimeOut.Q AND HMI_ValveControl.bWorkOn AND HMI_ValveControl.bSignalHome;

(*Error: Work position still active*)
ERROR_Valve.WorkFeedbackStillActive:=NOT(bInEstop) AND tonTimeOut.Q AND HMI_ValveControl.bHomeOn AND HMI_ValveControl.bSignalWork;

HMI_ValveControl.iErrorCode.0:=ERROR_Valve.NoWorkFeedback;
HMI_ValveControl.iErrorCode.1:=ERROR_Valve.NoHomeFeedback;
HMI_ValveControl.iErrorCode.2:=ERROR_Valve.HomeFeedbackStillActive;
HMI_ValveControl.iErrorCode.3:=ERROR_Valve.WorkFeedbackStillActive;

HMI_ValveControl.bError:=HMI_ValveControl.iErrorCode<>0;

(*Interlock*)
HMI_ValveControl.bInterlock:=bInEnable;

(************************************OUTPUTS**********************************************************************************)
(*Output Home*)
bOutCommandHome:=HMI_ValveControl.bHomeOn;

(*Output Work*)
bOutCommandWork:=HMI_ValveControl.bWorkOn;

(*Output Auto*)
bOutAuto:=(HMI_ValveControl.iMode=1);

(*Output error*)
bOutError:=HMI_ValveControl.bError;

END_FUNCTION_BLOCK

// ---- Base/Valve Control/POU/fcHMIBit.TcPOU
FUNCTION fcHMIBit : BOOL
VAR_INPUT
	bInToggle:BOOL;
	bInLatch:BOOL;
END_VAR
VAR_IN_OUT
	bHMI:BOOL;
	bPLC:BOOL;
END_VAR

(*set bPLC when bHMI set*)

IF bHMI AND NOT(bPLC) THEN
	bPLC:=1;
	bHMI:=0;
END_IF

END_FUNCTION

// ---- Base/Process Control/POU/POU.TcPOU
PROGRAM POU
VAR
		fbStateMachineCtrl:fbstepsequencer;
		step01Done:BOOL;
		step02Done:BOOL;
		step03Done:BOOL;
		step01Advance:BOOL;
		step01:stStep;
		step02:stStep;
		step03:stStep;
		step04:stStep;
		step05:stStep;
		step06:stStep;
		iCurrentStep:INT;
		lookuptable:fb1dLookup;
		aXvals: ARRAY [1..10] OF REAL :=[1,2,3,4,5,6,7,8,9,10]; (* Array of x values *)
		aYVals: ARRAY [1..10] OF REAL:=[3,9,12,11,14,16,18,19,21,23];	(* Array of x values *)
END_VAR

step01.tInStepDelay:=T#10S;
step02.tInStepDelay:=T#10S;
step03.tInStepDelay:=T#10S;
step04.tInStepDelay:=T#10S;
step05.tInStepDelay:=T#10S;
step06.tInStepDelay:=T#10S;

fbStateMachineCtrl(
	iInStep:=1 , 
	iInNextStep:=2 , 
	bInStepDone:=step01.bStepDone , 
	tInStepDelay:=step01.tInStepDelay , 
	bInStepMode:=step01.bInStepMode , 
	bInStepAdvance:=step01.bInStepAdvance , 
	bInit:= , 
	iInitStep:= 1, 
	bOutEnterEvent=>step01.bOutEnterEvent , 
	bOutExitEvent=>step01.bOutExitEvent ,
	bOutPaused=>step01.bOutPaused, 
	
	iOutCurrentStep=>iCurrentStep );

fbStateMachineCtrl(
	iInStep:= 2, 
	iInNextStep:=3 , 
	bInStepDone:=step02.bStepDone , 
	tInStepDelay:=step02.tInStepDelay , 
	bInStepMode:=step02.bInStepMode , 
	bInStepAdvance:=step02.bInStepAdvance , 
	bInit:= , 
	iInitStep:= 1, 
	bOutEnterEvent=>step02.bOutEnterEvent , 
	bOutExitEvent=>step02.bOutExitEvent , 
	bOutPaused=>step02.bOutPaused, 
	iOutCurrentStep=>iCurrentStep );

fbStateMachineCtrl(
	iInStep:= 3, 
	iInNextStep:=4 , 
	bInStepDone:=step03.bStepDone , 
	tInStepDelay:=step03.tInStepDelay , 
	bInStepMode:=step03.bInStepMode , 
	bInStepAdvance:=step03.bInStepAdvance , 
	bInit:= , 
	iInitStep:= 1, 
	bOutEnterEvent=>step03.bOutEnterEvent , 
	bOutExitEvent=>step03.bOutExitEvent , 
	bOutPaused=>step03.bOutPaused, 
	iOutCurrentStep=>iCurrentStep );

fbStateMachineCtrl(
	iInStep:= 4, 
	iInNextStep:=5 , 
	bInStepDone:=step04.bStepDone , 
	tInStepDelay:=step04.tInStepDelay , 
	bInStepMode:=step04.bInStepMode , 
	bInStepAdvance:=step04.bInStepAdvance , 
	bInit:= , 
	iInitStep:= 1, 
	bOutEnterEvent=>step04.bOutEnterEvent , 
	bOutExitEvent=>step04.bOutExitEvent , 
	bOutPaused=>step04.bOutPaused, 
	iOutCurrentStep=>iCurrentStep );

fbStateMachineCtrl(
	iInStep:= 5, 
	iInNextStep:=6 , 
	bInStepDone:=step05.bStepDone , 
	tInStepDelay:=step05.tInStepDelay , 
	bInStepMode:=step05.bInStepMode , 
	bInStepAdvance:=step05.bInStepAdvance , 
	bInit:= , 
	iInitStep:= 1, 
	bOutEnterEvent=>step05.bOutEnterEvent , 
	bOutExitEvent=>step05.bOutExitEvent , 
	bOutPaused=>step05.bOutPaused,
	iOutCurrentStep=>iCurrentStep );


fbStateMachineCtrl(
	iInStep:= 6, 
	iInNextStep:=1 , 
	bInStepDone:=step06.bStepDone , 
	tInStepDelay:=step06.tInStepDelay , 
	bInStepMode:=step06.bInStepMode , 
	bInStepAdvance:=step06.bInStepAdvance , 
	bInit:= , 
	iInitStep:= 1, 
	bOutEnterEvent=>step06.bOutEnterEvent , 
	bOutExitEvent=>step06.bOutExitEvent , 
	bOutPaused=>step06.bOutPaused,
	iOutCurrentStep=>iCurrentStep );
	
	
CASE fbStateMachineCtrl.iOutCurrentStep OF
	
END_CASE

lookuptable(x:= , xValues:= aXvals, yValues:=aYVals , y=> );

END_PROGRAM

// ---- Base/Process Control/POU/fbStepSequencer.TcPOU
FUNCTION_BLOCK fbStepSequencer
VAR_INPUT
	iInStep:		INT;	//Constant, the step which this block instance represents
	iInNextStep:	INT;	//Next step to go to when this step is done. Will be moved into iCurrentStep when bInStepDone is true
	bInStepDone:	BOOL;	//If true and iCurrentStep = iInStep, then we move to the next step.
	tInStepDelay:	TIME;	//Time between when the bInStepDone rises to when we move states, set to 0 to disable.
	bInStepMode:	BOOL;	//This input will pause the state machine at the completion of the current step until bInStepAdvance is set high. 
	bInStepAdvance:	BOOL;	//When the state machine is paused, this input will trigger the next step.
	bInit:			BOOL;	//Initializes the state machine to step iInitStep.
	iInitStep:		INT;	//Step that the machine will be initialized to when bInit is true. 
END_VAR
VAR_OUTPUT
	bOutEnterEvent:	BOOL;	//High for one scan when the state machine enters the state specified by iInStep for a single block usage.
	bOutExitEvent:	BOOL;	//High for one scan when the state machine leaves iInStep
	bOutPaused:		BOOL;	//Indicates if the sequencer is paused and waiting on a bInStepAdvance signal. 
	iOutCurrentStep:INT;	//Current state/step
END_VAR
VAR
	bNextStepCondition:BOOL;
	bMonitorState:BOOL;
	TONStepDelay:TON;
	
	tempbInStepDone:BOOL;
	tempbInStepAdvance:BOOL;
	tempbInStepMode:BOOL;
	temptInStepDelay:TIME;
	
	bBlipEnterEvent:BOOL;
	bBlipExitEvent: BOOL;
	tempiInitStep: INT;
END_VAR



IF  (iInStep = iOutCurrentStep) THEN
	
	(*Set bOutEnterEvent on first entry to state*)
	IF NOT bBlipEnterEvent THEN
		bBlipEnterEvent:=1;
		bOutEnterEvent:=1;
	ELSE
		bOutEnterEvent:=0;
	END_IF
	
	(*sample the input only when we are in current step as using the same instance function block*)
	temptInStepDelay:=tInStepDelay;				
	tempbInStepDone:=bInStepDone;
	tempbInStepAdvance:=bInStepAdvance;
	tempbInStepMode:=bInStepMode;
	tempiInitStep:=iInitStep;
	TONStepDelay.IN:=1;
	
	(*next step condition*)
	bNextStepCondition:=  TONStepDelay.Q AND(NOT(tempbInStepMode) OR (tempbInStepMode AND tempbInStepAdvance));
	
	bOutPaused :=  TONStepDelay.Q AND (tempbInStepMode AND NOT(tempbInStepAdvance));
	
	(*step complete map transition*)
	IF bNextStepCondition THEN
		TONStepDelay.IN:=0;              // reset step delay timer
		bBlipEnterEvent:=0;             //reset the one shot control for enter event
		bOutExitEvent:=1;				//Set only for one cycle 
		iOutCurrentStep:=iInNextStep;	//transition
	END_IF
	
ELSE
	bOutExitEvent:=0;
	bOutPaused :=  0;
END_IF

(*if binit received make initp step the state we move to*)
IF bInit THEN
		bInit:=0;
		iOutCurrentStep:=iInitStep;
END_IF

TONStepDelay(PT:=tInStepDelay);

END_FUNCTION_BLOCK

// ---- Base/Process Control/POU/fb1dLookup.TcPOU
FUNCTION_BLOCK fb1dLookup
VAR_INPUT
    x : REAL; (* Input value to lookup *)
    xValues : ARRAY [1..10] OF REAL; (* Array of x values *)
    yValues : ARRAY [1..10] OF REAL; (* Array of y values *)
END_VAR
VAR_OUTPUT
    y : REAL; (* Interpolated output value *)
END_VAR
VAR
    i : INT := 0; (* Index of the lower bound of the interpolation interval *)
    slope : REAL := 0.0; (* Slope of the interpolation interval *)
END_VAR

(* Perform the 1-d lookup *)
i := 1;
WHILE i < 10 AND x > xValues[i+1] DO
    i := i + 1;
END_WHILE

slope := (yValues[i+1] - yValues[i]) / (xValues[i+1] - xValues[i]);
y := yValues[i] + slope * (x - xValues[i]);

END_FUNCTION_BLOCK

// ---- Alarm System/POUs/02_Alarm_Handling/P_AlarmHandling.TcPOU
(**************************************************************************************
CopyRight Atlantis Operations UK Ltd 2015
AR500 Turbine Control System 

Program Purpose:
This program takes care of alarm handling and includes following functions:
	- sets a new alarm
	- resets not valid alarms
	- selects correct brake program if needed
	- selects operations associated with alarm 

Version history: Created with TwinCat V 2.11.2248
04/09/15	V 1.00	NSM - ODT First Release

Version history: Created with TwinCat V 2.9.0
19.01.2005	V 1.0.0	MLe
Initial Version
17.8.-24.8.2005 V 1.0.1 MLe
-Changes in alarm SMS; AlarmProgramAction, AddEmailToList
31.8.2005 V 1.0.2 MLe
-Service mode sms message comes trough in any circumstances
-Leading zeros added for time in sms message
8.9.2005 V 1.0.3 MLe
-\n changed to | as CfLf
6.10.2005 V 1.0.4 MLe
- 10 min Flow speed added to alarm SMS text
***************************************************************************************)

PROGRAM P_AlarmHandling
VAR
	arrAlarmSetDelay: ARRAY [1..1400] OF DINT;
	i: INT;
	arrAlarmResetDelay: ARRAY [1..1400] OF DINT;

	fbResets: FB_AlarmResets;
	bNoBrakeProgramSt: BOOL;
	(* AlarmProgramAction*)
	bEmailSentSt: BOOL;
	fbSendEmail: FB_SendEmail;										(* EN ABLED BY NM TEMPORARILY  *)
	bManuRstBrakePrgAlarmOnSt :BOOL;
	bNewAlarmSt: BOOL;
	bServiceModeBlockSt: BOOL;
	AlarmTime:TIMESTRUCT;

	(*Intouch communication*)


	WriteTime: BOOL;
	bGetTimeFlipFlop:BOOL;
	bGetTimeBusy:BOOL;
	bGetTimeErr: BOOL;
	iGetTimeErrId: DINT;

	(* Email for alarms *)
	arrEmailWaitList: ARRAY [1..5] OF STRING(255);
	iEmailPointer: INT := 0;
	bEmailSendingBusy: BOOL;
	sAlarmName: STRING(255);
	bStartEmailSending: BOOL;
	iEmailListCounter: INT;
	tonEmailDelay: TON;
	bSendEmailStartOff: BOOL;
	Step: INT := 10;
	tonSpaceDelay: TON;
	bDummy: BOOL;

	arrAlarmRepetitions: ARRAY [1..1400] OF ST_RepetitionArray;
	iRepetitionCntr: INT;
	iRemoveRepetitionCntr: INT;
	j: INT;

	alarmData: STRING(255);
	bFirstCycle: BOOL :=FALSE;
	rtrigManualReset: R_TRIG;

	tonFirstCycle: TON;

	TempCounter: INT;
	n: INT;
	TempCounterTest: INT;

	sTest: INT;

	iNumberOfAlarmsInHistory: INT := 200;

	k: INT;
	fbFileDelete: FB_FileDelete;
	bDelete_Busy: BOOL;
	bDelete_Error: BOOL;
	nDelete_ErrID: UDINT;
	fbFileDeleteOn: BOOL;

	sPreviousPathName				: T_MaxString ;	(* Set the previous Path name in the init program, added 15022010 MLe *)

	bFirstAlarmSetCycle: BOOL := TRUE;
	(*bFirstCycle2: BOOL;*)
	(*tonFirstCycle2: TON :=(PT:=t#1s);*)

	bInitComplete: BOOL;
	fbF_TRIG: F_TRIG;

	test: INT;
	tonCheckForEmails: TON;
	srSendEmailLatch: SR;
	bEngineerSendEmailTest: BOOL;
	ftrigEngineerSendEmailTest: F_TRIG;
END_VAR

(*TEMP ALARMS FOR TESTING*)
//P_ALARMS();
//P_Event_Logger();		For calling TC sysem events


(* Set new date for Alarm.txt file *)


ResetBrakePrograms();
bManuRstBrakePrgAlarmOnSt := FALSE; (* Reset before every loop *)

(* Reset repeating alarm *)
IF g_bOperAlarmManualReset THEN
	arrAlarms[a_bOperRepeatingAlarm].a := FALSE;
END_IF;

IF bFirstCycle THEN (* to avoid alarms with 0 time *)
	AlarmLoop();
END_IF;

(* 5 sec delay in a start up that Clock is synchronized *)
tonFirstCycle(IN:=TRUE , PT:= t#5.0s);
bFirstCycle:=tonFirstCycle.Q;


(* No Manu reset alarms with brake program on => New email can be sent when next preceding alarm occurs *)
IF NOT bManuRstBrakePrgAlarmOnSt THEN
	bEmailSentSt := FALSE;
END_IF;

TakeEmailFromList();
fbResets();

(* Delete previous Alarm.txt file *)
DeleteOldAlarmFile();

g_iOperAlarmStructSizeInBytes:=SIZEOF(arrAlarms[1]);
g_iOperIniStructSizeInBytes := SIZEOF(arrIni[1]);

P_AlarmTable();

ACTION ActiveShutdownAlarmCount:
(*NSM 231016*)
IF 	arrAlarms[i].b (*AND
	arrAlarms[i].eBrakeProgram < 99*)
THEN
	g_iOperErrorAlarmsActive := g_iOperErrorAlarmsActive  + 1;
END_IF
END_ACTION

ACTION AddEmailToList:
(* Add new alarm to email list to wait sending *)
IF iEmailPointer < 5 THEN

	(* Alarm short message includes: Park name, turbine name, brake program, alarm name, date and time.*)
	alarmData := CONCAT('"|Alarm|', g_sOperAlarmParkName);
	alarmData := CONCAT(alarmData, ' ');
	alarmData := CONCAT(alarmData, INT_TO_STRING(g_iOperAlarmParkId));
	alarmData := CONCAT(alarmData, '|');
	alarmData := CONCAT(alarmData, g_sOperAlarmTurbineName);
	alarmData := CONCAT(alarmData, ' ');
	alarmData := CONCAT(alarmData, INT_TO_STRING(g_iOperAlarmTurbineId));
	alarmData := CONCAT(alarmData, '|B');
	alarmData := CONCAT(alarmData, INT_TO_STRING(arrAlarms[i].eBrakeProgram));
	alarmData := CONCAT(alarmData, '|');
	alarmData := CONCAT(alarmData, arrAlarms[i].sName);

	(*alarmData := CONCAT(alarmData, '_');
	alarmData := CONCAT(alarmData, LEFT(REAL_TO_STRING(g_fOperFlowSpeedMean10minMe), 4)); (* Add Flow speed after alarm with 4 number *)
	alarmData := CONCAT(alarmData, 'm/s');*)

	alarmData := CONCAT(alarmData, '|B');
	alarmData := CONCAT(alarmData, INT_TO_STRING(arrAlarms[i].eBrakeProgram));
	alarmData := CONCAT(alarmData, '|');

	(* Leading zeros added for date*)
	IF arrAlarms[i].TimeOcc.wDay < 10 THEN
		alarmData := CONCAT(alarmData, CONCAT('0', WORD_TO_STRING(arrAlarms[i].TimeOcc.wDay)));
	ELSE
		alarmData := CONCAT(alarmData, WORD_TO_STRING(arrAlarms[i].TimeOcc.wDay));
	END_IF;
	alarmData := CONCAT(alarmData, '.');
	IF arrAlarms[i].TimeOcc.wMonth < 10 THEN
		alarmData := CONCAT(alarmData, CONCAT('0', WORD_TO_STRING(arrAlarms[i].TimeOcc.wMonth)));
	ELSE
		alarmData := CONCAT(alarmData, WORD_TO_STRING(arrAlarms[i].TimeOcc.wMonth));
	END_IF;
	alarmData := CONCAT(alarmData, '.');
	alarmData := CONCAT(alarmData, RIGHT (WORD_TO_STRING(arrAlarms[i].TimeOcc.wYear), 2));
	alarmData := CONCAT(alarmData, ' ');

(* Leading zeros added for time *)
	IF arrAlarms[i].TimeOcc.wHour < 10 THEN
		alarmData := CONCAT(alarmData, CONCAT('0', WORD_TO_STRING(arrAlarms[i].TimeOcc.wHour)));
	ELSE
		alarmData := CONCAT(alarmData, WORD_TO_STRING(arrAlarms[i].TimeOcc.wHour));
	END_IF;
	alarmData := CONCAT(alarmData, ':');
	IF	arrAlarms[i].TimeOcc.wMinute < 10 THEN
		alarmData := CONCAT(alarmData, CONCAT('0', WORD_TO_STRING(arrAlarms[i].TimeOcc.wMinute)));
	ELSE
		alarmData := CONCAT(alarmData, WORD_TO_STRING(arrAlarms[i].TimeOcc.wMinute));
	END_IF;
	alarmData := CONCAT(alarmData, '|');
	(* alarmData := CONCAT(alarmData, LEFT(REAL_TO_STRING(g_fOperFlowSpeedMean10minMe), 4)); (* Add Flow speed 251005 KKa *) 	DISABLED BY NIHAL MALIK *)
	alarmData := CONCAT(alarmData, ' m/s 10 min av.');
	alarmData := CONCAT(alarmData, '|');
(* Add reset mode *)
	IF arrAlarms[i].eResetMode=AUTO THEN
	alarmData := CONCAT(alarmData, 'AUTO reset mode ');
	ELSE
	alarmData := CONCAT(alarmData, 'MANUAL reset mode ');
	END_IF;
	alarmData := CONCAT(alarmData, '|');

(* Add fault comment *)

	alarmData := CONCAT(alarmData, 'Comment: ');
	alarmData := CONCAT(alarmData, arrAlarms[i].Comment);
	alarmData:= CONCAT(AlarmData,'|"');


(* Creating a subject to an email *)
	alarmData := CONCAT(alarmData, ' "Alarm Message from ');
//	alarmData:= CONCAT(AlarmData,stTurbineData.sOperAlarmParkName);	(*Action UPDATE This*)
	alarmData:= CONCAT(AlarmData,'"');
(*
(* Attach also a scopeViewFile *)
	alarmData := CONCAT(alarmData, ' "');
	alarmData:= CONCAT(AlarmData,stTurbineData.sOperScopeLocation);
	alarmData:= CONCAT(AlarmData,'"');
*)


	iEmailPointer := iEmailPointer + 1;
	arrEmailWaitList[iEmailPointer] := alarmData;

END_IF;
END_ACTION

ACTION AlarmAcknowledgement:
(* Alarm acknowledge *)(* 12012010 *)
	IF g_bOperAlarmManualResetREdge THEN
		IF arrAlarms[i].b THEN
			arrAlarms[i].iState := ActiveAcknowledged;(* Aktiivinen kuitattu *)
		ELSIF arrAlarms[i].iState = InactiveUnacknowledged THEN
			arrAlarms[i].iState := InactiveAcknowledged;(* Poistunut kuittaamaton => poistunut(kuitattu) *)
		ELSIF arrAlarms[i].iState = ActiveUnacknowledged    THEN(*12012010*)
			arrAlarms[i].iState := InactiveAcknowledged;
		END_IF
	END_IF

	IF ((arrAlarms[i].iState = ActiveUnacknowledged) AND (NOT arrAlarms[i].b)) THEN(*12012010*)
		arrAlarms[i].iState := InactiveUnacknowledged;
	ELSIF ((arrAlarms[i].iState = ActiveAcknowledged) AND (NOT arrAlarms[i].b)) THEN
		arrAlarms[i].iState := InactiveAcknowledged;
	END_IF
END_ACTION

ACTION AlarmBrake:
(* Set brake program *)
	IF arrAlarms[i].b = TRUE THEN
		CASE arrAlarms[i].eBrakeProgram OF

			B1:		g_bBrakeProg1Cmd := TRUE;
			B2:		g_bBrakeProg2Cmd := TRUE;
			B3:		g_bBrakeProg3Cmd := TRUE;
			B4:		g_bBrakeProg4Cmd := TRUE;
			B5:		g_bBrakeProg5Cmd := TRUE;
			B6:		g_bBrakeProg6Cmd := TRUE;
			B7:		g_bBrakeProg7Cmd := TRUE;
			B8:		g_bBrakeProg8Cmd := TRUE;
			B9:		g_bBrakeProg9Cmd := TRUE;
			B10:		g_bBrakeProg10Cmd := TRUE;
			B11:		g_bBrakeProg11Cmd := TRUE;
			B12:		g_bBrakeProg12Cmd := TRUE;
			B13:		g_bBrakeProg13Cmd := TRUE;
			B14:		g_bBrakeProg14Cmd := TRUE;
			B15:		g_bBrakeProg15Cmd := TRUE;
			B16:		g_bBrakeProg16Cmd := TRUE;
			B17:		g_bBrakeProg17Cmd := TRUE;
			B18:		g_bBrakeProg18Cmd := TRUE;
			B19:		g_bBrakeProg19Cmd := TRUE;
			B20:		g_bBrakeProg20Cmd := TRUE;
			B25:		g_bBrakeProg25Cmd := TRUE;
			B30:		g_bBrakeProg30Cmd := TRUE;
			B40:		g_bBrakeProg40Cmd := TRUE;

		ELSE
			bNoBrakeProgramSt := TRUE;
		END_CASE;
	END_IF;
END_ACTION

ACTION AlarmLoop:
(* Copy process values to right variables *)			(*NSM 231016*)
//MAIN_R();

(*Reset non end of tide shutdown alarms counter - NSM 31.10.16*)
g_iOperErrorAlarmsActive  := 0;

(*Reset count of number of active send email alarms*)(*Added NSM 28.9.17*)
g_iOperTurbine4SendEmailAlarmsActive := 0;

(* Do alarm actions *)
FOR i := 1 TO iMaxAlarms DO

	AlarmSet();
	AlarmRepetition();
	AlarmReset();
	AlarmBrake();
	AlarmProgramAction();
	AlarmParams();
	AlarmAcknowledgement();
	ActiveShutdownAlarmCount();
	SendEmail();

END_FOR;

//fbSCLogger.M_CheckEvent();
fbSCLogger();(*12012010*)
UpdateAlarmHistory();
bFirstAlarmSetCycle := FALSE;

(*If number of active send email alarms is > 0  then set flag to send email*)(*Added NSM 28.9.17*)
tonCheckForEmails(IN:=NOT tonCheckForEmails.Q, PT:=t#10s);

srSendEmailLatch(	SET1:= g_iOperTurbine4SendEmailAlarmsActive > 0,
					RESET:= g_iOperTurbine4SendEmailAlarmsActive = 0,
					Q1 => g_bOperTurbine4SendEmail	);

(*Added by NSM 20.02.18 to test alarm sending from SCADA*)
ftrigEngineerSendEmailTest(CLK:=bEngineerSendEmailTest);

IF 	FALSE AND	(*visu_bOperEnableTwinCAT_GUI	ACTION ADD LOGIC*)
	bEngineerSendEmailTest THEN
		g_bOperTurbine4SendEmail := TRUE;
ELSIF ftrigEngineerSendEmailTest.Q OR
		g_bOperOpModeService THEN			(*Added to stop emails being sent during pitching - NMS 26/06/18*)
		g_bOperTurbine4SendEmail := FALSE;
END_IF

(*IF g_iOperTurbine4SendEmailAlarmsActive > 0 THEN	(*Replaced above by NSM 25.10.17*)
		g_bOperTurbine4SendEmail := TRUE;
ELSE	g_bOperTurbine4SendEmail := FALSE;
END_IF*)
END_ACTION

ACTION AlarmParams:
(* Check the parameter limits for Set1 *)

	(* Check that Min is lower than Max *)
IF arrAlarms[i].param1.SetMin > arrAlarms[i].param1.SetMax THEN
arrAlarms[i].param1.SetMin:=arrAlarms[i].param1.SetMax;
END_IF;
	(* Check that set is lower than MAX *)
IF arrAlarms[i].Param1.Set >arrAlarms[i].param1.SetMax THEN
	arrAlarms[i].param1.Set := arrAlarms[i].param1.SetMax;
ELSE
	arrAlarms[i].param1.Set := arrAlarms[i].param1.Set;
END_IF;
	(* Check that set is higher than Min *)
IF arrAlarms[i].param1.Set < arrAlarms[i].param1.SetMin THEN
	arrAlarms[i].param1.Set := arrAlarms[i].param1.SetMin;
ELSE
arrAlarms[i].param1.Set :=  arrAlarms[i].param1.Set;

END_IF;

(* Check the parameter limits for Set2 *)

	(* Check that Min is lower than Max *)
IF arrAlarms[i].param2.SetMin > arrAlarms[i].param2.SetMax THEN
arrAlarms[i].param2.SetMin:=arrAlarms[i].param2.SetMax;
END_IF;
	(* Check that set is lower than Max *)
IF arrAlarms[i].Param2.Set >arrAlarms[i].param2.SetMax THEN
	arrAlarms[i].param2.Set := arrAlarms[i].param2.SetMax;
ELSE
	arrAlarms[i].param2.Set := arrAlarms[i].param2.Set;
END_IF;
	(* Check that set is higher than Min *)
IF arrAlarms[i].param2.Set < arrAlarms[i].param2.SetMin THEN
	arrAlarms[i].param2.Set := arrAlarms[i].param2.SetMin;
ELSE
arrAlarms[i].param2.Set :=  arrAlarms[i].param2.Set;

END_IF;
END_ACTION

ACTION AlarmProgramAction:
(* UPDATES MADE BY NSM ON 25/08/15 TO INCLUDE B99 WITH B100 GROUP *)

IF arrAlarms[i].b THEN
	(* Service mode is read directly from input, not from alarm *)
	(* Service mode blocks all emails *)
	(* Service mode announcement must come trough in any case *)
	(* IF ((NOT in_bOperOpModeService) OR (arrAlarms[i].sName = 'a_bOperServModeSt')) THEN *)
		(* Send email just once for alarms which have manual reset, brake program and email selection *)
		IF (arrAlarms[i].eResetMode = MANU) AND (NOT (arrAlarms[i].eBrakeProgram = B100)) AND (NOT (arrAlarms[i].eBrakeProgram = B99)) THEN (* Manual reset and brake program *)
			bManuRstBrakePrgAlarmOnSt := TRUE;(* Prevents consecutive alarms if stopping conditions are still valid *)
			IF (bNewAlarmSt AND (NOT bEmailSentSt) AND (arrAlarms[i].eAlarmProgram = Email)) THEN (* No email sent earlier and alarm program action is email *)
				AddEmailToList();
				bEmailSentSt := TRUE;
				(* Add alarm name to global variable for Scope View *)
				(* Prevent new alarm name as long as previous has been sent*) (*29012010*)
				IF g_sAlarmname = '' THEN
					g_sAlarmname:=arrAlarms[i].sName;
				END_IF
			END_IF;
		END_IF;
		(* Send email for alarms which do not have brake program but email selection; warnings and announcements....and
			also alarms which have auto reset send email if 'Email' selection is valid *)
		IF (arrAlarms[i].eBrakeProgram = B100) OR (arrAlarms[i].eBrakeProgram = B99) OR (arrAlarms[i].eResetMode = AUTO) THEN
				IF NOT(arrAlarms[i].eBrakeProgram = B100) AND NOT(arrAlarms[i].eBrakeProgram = B99) THEN
					IF bNewAlarmSt THEN
					(* Add alarm name to global variable for Scope View *)
					(* Prevent new alarm name as long as previous has been sent*) (*29012010*)
						IF g_sAlarmname = '' THEN
							g_sAlarmname:=arrAlarms[i].sName;
						END_IF
					END_IF;
				END_IF;
			IF (arrAlarms[i].eAlarmProgram = Email) THEN
				IF bNewAlarmSt THEN
					(* Add alarm name to global variable for Scope View *)
					(* Prevent new alarm name as long as previous has been sent*) (*29012010*)
					(* B100 alarms do not trigger scopeview file sending to server. That's why Alarmname cannot be set for them, 20100930 MLe *)
						 IF ((g_sAlarmname = '') AND (NOT(arrAlarms[i].eBrakeProgram = B100)) AND (NOT(arrAlarms[i].eBrakeProgram = B99))) THEN
							g_sAlarmname:=arrAlarms[i].sName;
						END_IF
					(* Service mode alarm must be sent every time it occurres *)
					IF ((NOT bEmailSentSt OR (arrAlarms[i].sName = 'a_bOperServModeSt')) AND (NOT arrAlarms[i].bRepetitionLimitExceeded)) THEN
						AddEmailToList();
					END_IF;
				END_IF;
			END_IF;
		END_IF;
	(* END_IF; *)
	bNewAlarmSt := FALSE;
END_IF;
END_ACTION

ACTION AlarmRepetition:
(*  Repeating alarm with AUTO reset causes special alarm.
    Repetition number 0 disables the whole function*)

IF (arrAlarms[i].eResetMode = AUTO) AND (arrAlarms[i].iRepetitionNumber <> 0) THEN

	(* Remove too old alarms from array , time period is minutes*)
	WHILE (((DT_TO_DWORD(SYSTEMTIME_TO_DT(g_stOperNTGetTime)) - arrAlarmRepetitions[i].arrRepetition[1]) / 60) > arrAlarms[i].iRepetitionPeriod) AND (arrAlarmRepetitions[i].arrRepetition[1] <> 0) DO
		(* Move every alarm time one step further *)
		iRemoveRepetitionCntr := 1;
		WHILE ((arrAlarmRepetitions[i].arrRepetition[iRemoveRepetitionCntr + 1] <> 0) AND (iRemoveRepetitionCntr < 10)) DO
			arrAlarmRepetitions[i].arrRepetition[iRemoveRepetitionCntr] := arrAlarmRepetitions[i].arrRepetition[iRemoveRepetitionCntr + 1];
			iRemoveRepetitionCntr :=  iRemoveRepetitionCntr + 1;
		END_WHILE;
		arrAlarmRepetitions[i].arrRepetition[iRemoveRepetitionCntr] := 0;
	END_WHILE;


	(* Count old repeated alarms. iRepetitionCntr points to first  unoccupied place in array *)
	iRepetitionCntr := 1;
	WHILE (arrAlarmRepetitions[i].arrRepetition[iRepetitionCntr] <> 0) DO
		iRepetitionCntr := iRepetitionCntr + 1;
	END_WHILE;

	(* Add  new alarm time to array *)
	IF bNewAlarmSt AND  (iRepetitionCntr < 11) THEN
		arrAlarmRepetitions[i].arrRepetition[iRepetitionCntr] := DT_TO_DWORD(SYSTEMTIME_TO_DT(g_stOperNTGetTime));
		iRepetitionCntr := iRepetitionCntr + 1;
	END_IF


	(* If repetitions are equal to limit value then set 'Repeating error' on and mark the alarm which caused the error.*)
	IF (iRepetitionCntr > 1) THEN
		IF ((iRepetitionCntr - 1) >= arrAlarms[i].iRepetitionNumber) THEN
			arrAlarms[a_bOperRepeatingAlarm].a := TRUE;
			arrAlarms[i].bRepetitionLimitExceeded := TRUE;
		END_IF;
	END_IF;

END_IF;
END_ACTION

ACTION AlarmReset:
(* UPDATED BY NSM ON 25/08/15 TO INCLUDE B99 BRAKE PROGRAM FOR RESETS AND IDLE STATE REMOVED *)
(* UPDATED BY NSM ON 01/12/16 TO REINSTATE ORIGINAL APPROACH TO RESETTING THESE ALARMS *)
(* Alarm Resetting *)

	(*AUTO*)
	IF arrAlarms[i].eResetMode = AUTO THEN
		(* No active alarm *)
		IF 	(arrAlarms[i].b AND  (NOT arrAlarms[i].a)) 
			(* No brake program or machine stopped => enable reset count *)
				(*g_eMainState = STOP OR
				g_eMainState = SAFETY_TRIPPED*)  (*action re-instate make it less spaghetti code*)
		(*	(	(arrAlarms[i].eBrakeProgram = B100) OR
				(arrAlarms[i].eBrakeProgram = B99) OR
				g_bOperMaStStopSt OR
				g_bOperMaStIdleSt OR			///ACTION Re enable to state mc when built
				g_bOperMaStStandbySt		)*)
				
		THEN
			arrAlarmResetDelay[i] := arrAlarmResetDelay[i] + g_iOperCycleTime;
			(* If time elapsed then reset alarm *)
			IF arrAlarmResetDelay[i] >= (arrAlarms[i].iResetDelay  * 100) THEN
				arrAlarms[i].b := FALSE;
			ELSE
				arrAlarms[i].b := TRUE;
			END_IF;
		(* Alarm is active or there has not been alarm *)
		ELSE
			arrAlarmResetDelay[i] := 0; (* Alarm activated again or no alarm *)
		END_IF;

		(* Reset repeating error  *)
		IF arrAlarms[i].bRepetitionLimitExceeded AND g_bOperAlarmManualReset THEN
			arrAlarms[i].bRepetitionLimitExceeded := FALSE;
			FOR j := 1 TO 10 DO
				arrAlarmRepetitions[i].arrRepetition[j] := 0;
			END_FOR;
		END_IF;
	ELSE

	(*MANU*)
		(* No active alarm *)
		IF (arrAlarms[i].b) AND (NOT arrAlarms[i].a)  THEN
			(* Non Safety Alarm without brake program OR machine stopped OR Idling mode On AND manual reset *)

(*Removed by NSM on 17/03/16*)
(*arrAlarms[i].eBrakeProgram = B100 OR arrAlarms[i].eBrakeProgram = B99 OR *)

			IF 	(*(g_bOperMaStStopSt OR g_bOperMaStIdleSt OR g_bOperMaStStandbySt) AND*) g_bOperAlarmManualResetREdge AND arrAlarms[i].eBrakeProgram > 10 THEN
				arrAlarms[i].b := FALSE;

			ELSIF (*NOT(g_bOperMaStNormalStopSt OR g_bOperMaStEmergencyStopSt) AND *) g_bOperAlarmManualResetREdge AND (arrAlarms[i].eBrakeProgram = 99 OR arrAlarms[i].eBrakeProgram = 100) THEN
				arrAlarms[i].b := FALSE;
			(* Safety Alarm Manual Reset *)
(*			ELSIF (g_bOperMaStStopSt OR g_bOperMaStIdleSt) AND arrAlarms[i].eBrakeProgram < 10 AND g_bOperAlarmManualSafetyResetREdge THEN	*)
			ELSIF (*(g_bOperMaStStopSt OR g_bOperMaStIdleSt) AND*) g_bOperAlarmManualSafetyResetREdge THEN
				arrAlarms[i].b := FALSE;
			END_IF;
		END_IF;
	END_IF;

	(*Alarm Disabled*)
		(* No active alarm *)
		IF (arrAlarms[i].b) AND (NOT arrAlarms[i].Enable)  THEN
			(* Alarm disabled AND manual reset *)
			(*IF 	(NOT arrAlarms[i].Enable) AND (g_bOperAlarmManualReset THEN	*)(*Replcaed by NSM 28.05.16*)
			IF 	(NOT arrAlarms[i].Enable) AND (g_bOperAlarmManualResetREdge OR g_bOperAlarmManualSafetyResetREdge) THEN
				arrAlarms[i].b := FALSE;
				arrAlarms[i].iState := InactiveAcknowledged;(*12012010*)
			END_IF;
		END_IF;


	arrAlarms[i].iResetDelayElapsed := arrAlarmResetDelay[i]/100;

            arrAlarmStatus[i] := arrAlarms[i].b;
			 arrAlarmGroup[i] := arrAlarms[i].iGroup;
            arrAlarmGroup[i] := arrAlarms[i].iGroup;
END_ACTION

ACTION AlarmSet:
(* Alarm Setting *)
(*========== START OF FUNCTION_BLOCK / PROGRAMM ============*)
 arrAlarms[i].eBrakeProgram;
(* INHIBIT SC  LOGGER UNTIL INIT COMPLETE - 09/02/17  AG. *)
fbF_TRIG(CLK:=g_bOperMaStInitSt);


IF fbF_TRIG.Q THEN
	bInitComplete:=TRUE;
END_IF

	(* In case of PLC restart old b-alarms have to be picked up to alarm screen *)
	IF bFirstAlarmSetCycle AND arrAlarms[i].b AND arrAlarms[i].Enable THEN
		(* Copy old b-alarms to history *)
					(*n:=1;*)
					FOR n := 1 TO iNumberOfAlarmsInHistory - 1 DO
						arrLastAlarms[iNumberOfAlarmsInHistory + 1 - n] := arrLastAlarms[iNumberOfAlarmsInHistory - n];
					END_FOR;
					arrLastAlarms[1]:=arrAlarms[i];
					arrLastAlarms[1].Index:=i;
	END_IF


	(* Normal case *)
	IF (arrAlarms[i].a AND (NOT arrAlarms[i].b) AND arrAlarms[i].Enable)  THEN (* Enable condition added *)
		IF arrAlarmSetDelay[i]  >= (arrAlarms[i].iSetDelay * 100) THEN
			arrAlarms[i].b := TRUE;
			bNewAlarmSt := TRUE; (*Send email if needed *)
			arrAlarms[i].sTimeOcc := gsLocalSystemTime;
			arrAlarms[i].TimeOcc := g_stOperNTGetTime;
			arrAlarms[i].iState := ActiveUnacknowledged; (* 12012010 *)
			(* Process variables *)
			arrAlarms[i].stProcessVariables.fGeneratorSpeed :=0; (* g_fOperGenSpeedFromConverterRpmMe;	*)	(*NSM 231016*)
			arrAlarms[i].stProcessVariables.fPitchAngle := 0(*g_fPitchAngleFilteredDeg*);	
			arrAlarms[i].stProcessVariables.fPower := 0(*g_fOperGenPowerFromConverterMe*);
			arrAlarms[i].stProcessVariables.fFlowSpeed := 0(*g_fOperFlowSpeed10minAverage*);


				IF arrAlarms[i].b  AND arrAlarms[i].eBrakeProgram<=40  THEN   (* A.G. Inhibit call when brake prog LEQ  40*)
					(* Call status code logger *)
					


					(* Make a buffer of statuscodes for HMI ********************)
					(* Copy a new alarm to history *)
					(*n:=1;*)
					FOR n := 1 TO iNumberOfAlarmsInHistory - 1 DO
						arrLastAlarms[iNumberOfAlarmsInHistory + 1 - n] := arrLastAlarms[iNumberOfAlarmsInHistory - n];
					END_FOR;
					arrLastAlarms[1]:=arrAlarms[i];
					arrLastAlarms[1].Index:=i;

					(* Make a buffer of statuscodes for HMI ********************)

				END_IF

		ELSE
			arrAlarms[i].b := FALSE;
		END_IF;
		arrAlarmSetDelay[i] := arrAlarmSetDelay[i] + g_iOperCycleTime;
	ELSE arrAlarmSetDelay[i] := 0;

	END_IF
	arrAlarms[i].iSetDelayElapsed := arrAlarmSetDelay[i]/100;
END_ACTION

ACTION DeleteOldAlarmFile:
(* If a new day detected then delete an old alarm file in directory \Hard Disk\DAT\Transfer' *)
(* A presumption is that file has been already copied to D:\DAT *)
(* The FB shows error 1804 if directory is empty *)

IF  (sPreviousPathName <> gsSC_PathName) OR fbFileDeleteOn THEN

	fbFileDeleteOn := TRUE;

	fbFileDelete(
		sNetId:='',
		sPathName:= sPreviousPathName,
		ePath:= PATH_GENERIC,
		bExecute:= TRUE,
		tTimeout:= t#5s,
		bBusy=> bDelete_Busy,
		bError=> bDelete_Error,
		nErrId=> nDelete_ErrID);
	
	IF NOT fbFileDelete.bBusy THEN
		fbFileDelete(bExecute := FALSE);
		fbFileDeleteOn := FALSE;
	END_IF

END_IF

sPreviousPathName := gsSC_PathName;
END_ACTION

ACTION ResetBrakePrograms:
g_bBrakeProg1Cmd := FALSE;
g_bBrakeProg2Cmd := FALSE;
g_bBrakeProg3Cmd := FALSE;
g_bBrakeProg4Cmd := FALSE;
g_bBrakeProg5Cmd := FALSE;
g_bBrakeProg6Cmd := FALSE;
g_bBrakeProg7Cmd := FALSE;
g_bBrakeProg8Cmd := FALSE;
g_bBrakeProg9Cmd := FALSE;
	(* These need a different group to reset *)
g_bBrakeProg10Cmd := FALSE;
g_bBrakeProg11Cmd := FALSE;
g_bBrakeProg12Cmd := FALSE;
g_bBrakeProg13Cmd := FALSE;
g_bBrakeProg14Cmd := FALSE;
g_bBrakeProg15Cmd := FALSE;
g_bBrakeProg16Cmd := FALSE;
g_bBrakeProg17Cmd := FALSE;
g_bBrakeProg18Cmd := FALSE;
g_bBrakeProg19Cmd := FALSE;
g_bBrakeProg20Cmd := FALSE;
g_bBrakeProg25Cmd := FALSE;
g_bBrakeProg30Cmd := FALSE;
g_bBrakeProg40Cmd := FALSE;
bNoBrakeProgramSt := FALSE;
END_ACTION

ACTION SendEmail:
(*Added by NSM to count number of alarms that want to send emails - 28.9.17*)

IF 	(*arrAlarms[i].eAlarmProgram = 1 AND*)(*ACTION: Set this up to use the correct attribute of an alarm from the excel sheet*)
	arrAlarms[i].b AND
	arrAlarms[i].eBrakeProgram <= 40 
THEN
	g_iOperTurbine4SendEmailAlarmsActive := g_iOperTurbine4SendEmailAlarmsActive + 1;
END_IF
END_ACTION

ACTION TakeEmailFromList:
CASE Step OF

	10:		IF iEmailPointer > 0 THEN
				Step := 20;(* Send alarm *)
			ELSE
				Step := 30;(* 'Send' empty string *)
			END_IF;

			(* Alarm from wait list *)
	20:		sAlarmName := arrEmailWaitList[1];
			bStartEmailSending := TRUE;
			iEmailListCounter := 1;
			WHILE (iEmailListCounter < 5) AND (arrEmailWaitList[iEmailListCounter] <> '') DO
				arrEmailWaitList[iEmailListCounter] := arrEmailWaitList[iEmailListCounter + 1];
				iEmailListCounter := iEmailListCounter + 1;
			END_WHILE;
			iEmailPointer := iEmailPointer - 1;
			IF iEmailPointer < 0 THEN
				iEmailPointer := 0;
			END_IF;
			bDummy := TRUE;
			Step := 50;

			(* Reset sending ( bStartEmailSending := FALSE)*)
	30:		sAlarmName := '';
			bStartEmailSending := FALSE;
			Step := 50;

			(* Every second NT_StartProcess always fails, so that dummy alarm must be sent *)
	35:		sAlarmName := 'DUMMY';
			bStartEmailSending := TRUE;
			Step := 50;

	50:		fbSendEmail(sAlarmName:= sAlarmName, bStart:= bStartEmailSending , bNTProcessBusy=> bEmailSendingBusy);
			IF sAlarmName = '' THEN
				Step := 70;(* Set delay for NT_StartProcess after empty string *)
			ELSE
				Step := 60;(* Set delay for NT_StartProcess after alarm*)
			END_IF;

			(* Delay after sending *)
	60:		tonEmailDelay(IN:=NOT  tonEmailDelay.Q, PT:= T#1s, Q=> , ET=> );
			IF tonEmailDelay.Q THEN
				Step := 30;
			END_IF;

			(* Delay after reseting *)
	70:		tonSpaceDelay(IN:=NOT  tonSpaceDelay.Q, PT:= T#1s, Q=> , ET=> );
			IF tonSpaceDelay.Q THEN
				IF bDummy  THEN
					Step := 35;
					bDummy := FALSE;
				ELSE
					Step := 10;
				END_IF;
			END_IF;

END_CASE;
END_ACTION

ACTION UpdateAlarmHistory:
(*12012010*)
 (* Updating the statuscode attributes in the history *)
FOR k := 1 TO iNumberOfAlarmsInHistory DO

	IF arrLastAlarms[k].Index = 0 THEN
		EXIT;(* It's no use to check further since there are no alarms *)
	ELSE
		IF arrLastAlarms[k].iState = ActiveUnacknowledged THEN
			arrLastAlarms[k].iResetDelayElapsed:=arrAlarms[arrLastAlarms[k].Index].iResetDelayElapsed;
		END_IF
	END_IF

	(* Change status in history array based on status in current alarm array *)
	IF (arrLastAlarms[k].iState = ActiveUnacknowledged)  AND ((arrAlarms[arrLastAlarms[k].Index].iState = ActiveAcknowledged) OR
	(arrLastAlarms[k].sTimeOcc <> arrAlarms[arrLastAlarms[k].Index].sTimeOcc)) THEN
		arrLastAlarms[k].iState := ActiveAcknowledged;
	ELSIF (arrLastAlarms[k].iState = InactiveUnacknowledged)  AND arrAlarms[arrLastAlarms[k].Index].iState = InactiveAcknowledged THEN
		arrLastAlarms[k].iState := InactiveAcknowledged;
	ELSIF (arrLastAlarms[k].iState = ActiveUnacknowledged)  AND arrAlarms[arrLastAlarms[k].Index].iState = InactiveUnacknowledged THEN
		arrLastAlarms[k].iState := InactiveUnacknowledged;
	ELSIF (arrLastAlarms[k].iState = ActiveAcknowledged)  AND arrAlarms[arrLastAlarms[k].Index].iState = InactiveAcknowledged THEN
		arrLastAlarms[k].iState := InactiveAcknowledged;
	ELSIF (arrLastAlarms[k].iState = ActiveUnacknowledged)  AND arrAlarms[arrLastAlarms[k].Index].iState = InactiveAcknowledged THEN
		arrLastAlarms[k].iState := InactiveAcknowledged;
	END_IF

END_FOR;
END_ACTION

END_PROGRAM

// ---- Alarm System/POUs/02_Alarm_Handling/FB_AlarmResets.TcPOU
FUNCTION_BLOCK FB_AlarmResets
VAR_INPUT
END_VAR
VAR_OUTPUT
END_VAR
VAR
	//ACTION THIS SHOULD BE A PRPGRAM AND NOT A FUNCTION BLOCK. USING GLOBAL VARS

	ManualAlarmReset:	TP;			(* One second pulse for manual alarm reset *)
	AutomaticReset:	TP;			(*    One second pulse for automatic alarm reset, only in stop mode every e.g. 10 seconds *)
	AutomaticResetTiming: TON; 	(* Interval timer for automatic resets*)
	rtrigManualReset: R_TRIG;
	TPResetAfterGridFailure: TP;
	TONResetAfterGridFailure: TON;
	rtrigManualSafetyReset: R_TRIG;
	SafetyAlarmReset: TP;
END_VAR

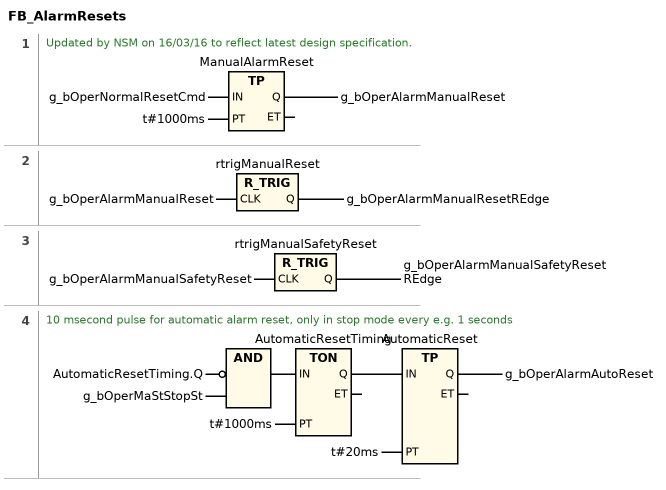
// NETWORK 1
// 					Updated by NSM on 16/03/16 to reflect latest design specification.
//
//
//
//
ManualAlarmReset(IN := g_bOperNormalResetCmd, PT := t#1000ms); // TP
g_bOperAlarmManualReset := ManualAlarmReset.Q;

// NETWORK 2
rtrigManualReset(CLK := g_bOperAlarmManualReset); // R_TRIG
g_bOperAlarmManualResetREdge := rtrigManualReset.Q;

// NETWORK 3
rtrigManualSafetyReset(CLK := g_bOperAlarmManualSafetyReset); // R_TRIG
g_bOperAlarmManualSafetyResetREdge := rtrigManualSafetyReset.Q;

// NETWORK 4
// 10 msecond pulse for automatic alarm reset, only in stop mode every e.g. 1 seconds
AutomaticResetTiming(IN := NOT AutomaticResetTiming.Q AND g_bOperMaStStopSt, PT := t#1000ms); // TON
AutomaticReset(IN := AutomaticResetTiming.Q, PT := t#20ms); // TP
g_bOperAlarmAutoReset := AutomaticReset.Q;

END_FUNCTION_BLOCK

// ---- Alarm System/POUs/02_Alarm_Handling/FB_SendEmail.TcPOU
FUNCTION_BLOCK FB_SendEmail
VAR_INPUT
	sAlarmName: STRING(255);
	bStart: BOOL;
END_VAR
VAR_OUTPUT
	bNTProcessBusy:BOOL;
END_VAR
VAR
	NT_StartProcess: NT_StartProcess;
	sPath: STRING := 'C:\DAT\ExecutableFiles\Sendemail.bat ';
	sPath2: STRING := 'C:\DAT\ExecutableFiles';
	bNTErr: BOOL;

	dummy: BOOL;
END_VAR

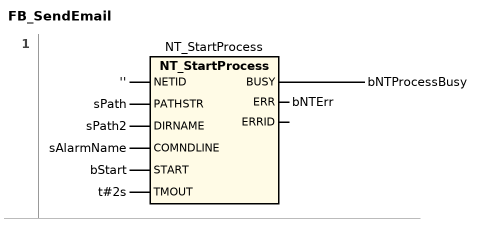
// NETWORK 1
NT_StartProcess(
    NETID := '',
    PATHSTR := sPath,
    DIRNAME := sPath2,
    COMNDLINE := sAlarmName,
    START := bStart,
    TMOUT := t#2s,
    ERR => bNTErr);
bNTProcessBusy := NT_StartProcess.BUSY;

END_FUNCTION_BLOCK

// ---- Alarm System/POUs/02_Alarm_Handling/P_AlarmTable.TcPOU
PROGRAM P_AlarmTable
VAR
	iCheckTestAlarms : UINT;
	iCount_B17: UINT;
	iCount_B1: UINT;
	iCount_B9: UINT;
	iCount_B14: UINT;
	iCount_B4: UINT;
	iCount_B5: UINT;
	iCount_B2: UINT;
	iCount_B20: UINT;
	iCount_B99: UINT;
	iTotalBrakeAlarms:	UINT;
	arrAlarmsTableB9: ARRAY [1..20] OF UINT;
	arrAlarmsTableB9_names: ARRAY [1..20] OF STRING;
	arrAlarmsTableB1: ARRAY [1..20] OF UINT;
	arrAlarmsTableB1_names: ARRAY [1..20] OF STRING;
	arrAlarmsTableB17: ARRAY [1..20] OF UINT;
	arrAlarmsTableB17_names: ARRAY [1..20] OF STRING;
	arrAlarmsTableB4: ARRAY [1..20] OF UINT;
	arrAlarmsTableB4_names: ARRAY [1..20] OF STRING;
	arrAlarmsTableB14: ARRAY [1..20] OF UINT;
	arrAlarmsTableB14_names: ARRAY [1..20] OF STRING;
	arrAlarmsTableB2: ARRAY [1..20] OF UINT;
	arrAlarmsTableB2_names: ARRAY [1..20] OF STRING;
	arrAlarmsTableB20: ARRAY [1..20] OF UINT;
	arrAlarmsTableB20_names: ARRAY [1..20] OF STRING;
	arrAlarmsTableB5: ARRAY [1..20] OF UINT;
	arrAlarmsTableB5_names: ARRAY [1..20] OF STRING;
	arrAlarmsTableB99: ARRAY [1..20] OF UINT;
	arrAlarmsTableB99_names: ARRAY [1..20] OF STRING;
END_VAR

iCount_B17 := 0;
iCount_B1 := 0;
iCount_B14 := 0;
iCount_B4 := 0;
iCount_B9 := 0;
iCount_B5 := 0;
iCount_B2 := 0;
iCount_B20 := 0;
iCount_B99 := 0;
MEMSET( ADR( arrAlarmsTableB1 ), 0, SIZEOF( arrAlarmsTableB1 ) );
MEMSET( ADR( arrAlarmsTableB1_names ), 0, SIZEOF( arrAlarmsTableB1_names ) );
MEMSET( ADR( arrAlarmsTableB17 ), 0, SIZEOF( arrAlarmsTableB17 ) );
MEMSET( ADR( arrAlarmsTableB17_names ), 0, SIZEOF( arrAlarmsTableB17_names ) );

MEMSET( ADR( arrAlarmsTableB4 ), 0, SIZEOF( arrAlarmsTableB4 ) );
MEMSET( ADR( arrAlarmsTableB4_names ), 0, SIZEOF( arrAlarmsTableB4_names ) );

MEMSET( ADR( arrAlarmsTableB14 ), 0, SIZEOF( arrAlarmsTableB14 ) );
MEMSET( ADR( arrAlarmsTableB14_names ), 0, SIZEOF( arrAlarmsTableB14_names ) );
MEMSET( ADR( arrAlarmsTableB9 ), 0, SIZEOF( arrAlarmsTableB9 ) );
MEMSET( ADR( arrAlarmsTableB9_names ), 0, SIZEOF( arrAlarmsTableB9_names ) );
MEMSET( ADR( arrAlarmsTableB5 ), 0, SIZEOF( arrAlarmsTableB5 ) );
MEMSET( ADR( arrAlarmsTableB5_names ), 0, SIZEOF( arrAlarmsTableB5_names ) );
MEMSET( ADR( arrAlarmsTableB2 ), 0, SIZEOF( arrAlarmsTableB2 ) );
MEMSET( ADR( arrAlarmsTableB2_names ), 0, SIZEOF( arrAlarmsTableB2_names ) );

MEMSET( ADR( arrAlarmsTableB20 ), 0, SIZEOF( arrAlarmsTableB20 ) );
MEMSET( ADR( arrAlarmsTableB20_names ), 0, SIZEOF( arrAlarmsTableB20_names ) );

MEMSET( ADR( arrAlarmsTableB99 ), 0, SIZEOF( arrAlarmsTableB99 ) );
MEMSET( ADR( arrAlarmsTableB99_names ), 0, SIZEOF( arrAlarmsTableB99_names ) );

FOR iCheckTestAlarms := 1 TO iMaxAlarms DO

	IF  arrAlarms[iCheckTestAlarms].eBrakeProgram = 17 AND arrAlarms[iCheckTestAlarms].b THEN
		iCount_B17 := iCount_B17 + 1;
		arrAlarmsTableB17[iCount_B17] := iCheckTestAlarms;
		arrAlarmsTableB17_names[iCount_B17] := arrAlarms[iCheckTestAlarms].sName;
		
	ELSIF  arrAlarms[iCheckTestAlarms].eBrakeProgram = 1 AND arrAlarms[iCheckTestAlarms].b THEN
		iCount_B1 := iCount_B1 + 1;
		arrAlarmsTableB1[iCount_B1] := iCheckTestAlarms;
		arrAlarmsTableB1_names[iCount_B1] := arrAlarms[iCheckTestAlarms].sName;
		
	ELSIF  arrAlarms[iCheckTestAlarms].eBrakeProgram = 4 AND arrAlarms[iCheckTestAlarms].b THEN
		iCount_B4 := iCount_B4 + 1;
		arrAlarmsTableB4[iCount_B4] := iCheckTestAlarms;
		arrAlarmsTableB4_names[iCount_B4] := arrAlarms[iCheckTestAlarms].sName;	
		
	ELSIF  arrAlarms[iCheckTestAlarms].eBrakeProgram = 14 AND arrAlarms[iCheckTestAlarms].b THEN
		iCount_B14 := iCount_B14 + 1;
		arrAlarmsTableB14[iCount_B14] := iCheckTestAlarms;
		arrAlarmsTableB14_names[iCount_B14] := arrAlarms[iCheckTestAlarms].sName;

	ELSIF  arrAlarms[iCheckTestAlarms].eBrakeProgram = 9 AND arrAlarms[iCheckTestAlarms].b THEN
			iCount_B9 := iCount_B9 + 1;
			arrAlarmsTableB9[iCount_B9] := iCheckTestAlarms;
			arrAlarmsTableB9_names[iCount_B9] := arrAlarms[iCheckTestAlarms].sName;
	
	ELSIF  arrAlarms[iCheckTestAlarms].eBrakeProgram = 5 AND arrAlarms[iCheckTestAlarms].b THEN
			iCount_B5 := iCount_B5 + 1;
			arrAlarmsTableB5[iCount_B5] := iCheckTestAlarms;
			arrAlarmsTableB5_names[iCount_B5] := arrAlarms[iCheckTestAlarms].sName;

	ELSIF  arrAlarms[iCheckTestAlarms].eBrakeProgram = 2 AND arrAlarms[iCheckTestAlarms].b THEN
		iCount_B2 := iCount_B2 + 1;
		arrAlarmsTableB2[iCount_B2] := iCheckTestAlarms;
		arrAlarmsTableB2_names[iCount_B2] := arrAlarms[iCheckTestAlarms].sName;
		
	ELSIF  arrAlarms[iCheckTestAlarms].eBrakeProgram = 20 AND arrAlarms[iCheckTestAlarms].b THEN
		iCount_B20 := iCount_B20 + 1;
		arrAlarmsTableB20[iCount_B20] := iCheckTestAlarms;
		arrAlarmsTableB20_names[iCount_B20] := arrAlarms[iCheckTestAlarms].sName;


	ELSIF  arrAlarms[iCheckTestAlarms].eBrakeProgram = 99 AND arrAlarms[iCheckTestAlarms].b THEN
		iCount_B99 := iCount_B99 + 1;
		arrAlarmsTableB99[iCount_B99] := iCheckTestAlarms;
		arrAlarmsTableB99_names[iCount_B99] := arrAlarms[iCheckTestAlarms].sName;

	END_IF

END_FOR

	iTotalBrakeAlarms	:=iCount_B1 + iCount_B2 + iCount_B9;

END_PROGRAM

// ---- Alarm System/TC3 EventLogger/MultipleAlarmCreation.TcPOU
PROGRAM MultipleAlarmCreation
VAR
	bIsInitalized : BOOL;
    fbAlarm : ARRAY[1..10] OF FB_TcAlarm;
    bRaiseAlarm : ARRAY[1..10] OF BOOL;;
    bClearAlarm : BOOL;
	bConfirmAlarm:BOOL; 
    fbSourceInfo : FB_TcSourceInfo;
	index:USINT;
END_VAR

IF NOT bIsInitalized THEN
    bIsInitalized := TRUE;
    fbSourceInfo.Clear();
    fbSourceInfo.sName := 'Water pump 3';
    fbAlarm[1].CreateEx(TC_Events.AlarmSystem.B99, FALSE, fbSourceInfo);
	fbAlarm[2].CreateEx(TC_Events.AlarmSystem.B20, FALSE, fbSourceInfo);
	fbAlarm[3].CreateEx(TC_Events.AlarmSystem.B20, FALSE, fbSourceInfo);
END_IF

IF bRaiseAlarm[1] THEN
    bRaiseAlarm[1] := FALSE;
    fbAlarm[1].ipArguments.Clear().AddString('Water Pump1');
    fbAlarm[1].Raise(0);
END_IF

IF bRaiseAlarm[2] THEN
    bRaiseAlarm[2] := FALSE;
    fbAlarm[2].ipArguments.Clear().AddString('B20 instance 1');
    fbAlarm[2].Raise(0);
END_IF

IF bRaiseAlarm[3] THEN
    bRaiseAlarm[3] := FALSE;
    fbAlarm[3].ipArguments.Clear().AddString('B20 instance 2');
    fbAlarm[3].Raise(0);
END_IF

(*
IF bConfirmAlarm THEN
    bConfirmAlarm := FALSE;
    fbAlarm.Confirm(0);
END_IF
*)

IF bClearAlarm THEN
	FOR index:=1 TO 3 DO
		 fbAlarm[index].Clear(0, TRUE);
	END_FOR
   // bClearAlarm := FALSE;
   
END_IF

END_PROGRAM

// ---- Alarm System/TC3 EventLogger/P_EventLogger_TCSAlarms.TcPOU
PROGRAM P_EventLogger_TCSAlarms

//CREATES AND HANDLES ALARMS BASED ON THE WIN WIND ALARM STRUCTURE THAT EXISTS ALREADY
VAR
	fbAlarm:ARRAY[1..222] OF FB_TcAlarm;
	fbSourceInfo : FB_TcSourceInfo;
	binit: BOOL;
	i:UINT; 
	index2:UINT;
END_VAR

initAlarms();
IF bInit THEN
	FOR index2:=1 TO 222 DO
		RaiseAlarms();
		
		ClearAlarms();
	END_FOR
END_IF

ACTION ClearAlarms:
// IF WIN WIND ALARM IS CLEARED, COMMAND THE INSTANCE OF THE CREATE TC3 ALARM TO CLEAR ALSO
IF NOT arrAlarms[index2].b THEN
	 fbAlarm[index2].Clear(0, TRUE);
END_IF
END_ACTION

ACTION initAlarms:
//Initialise alarms based on the brake program defined in the arrAlarms array of ST_ALARMSTRUCTURE
IF NOT binit THEN
	FOR i:=1 TO 222 DO
		CASE arrAlarms[i].eBrakeProgram OF
			B1:
				fbSourceInfo.Clear();
				fbSourceInfo.sName := arrAlarms[i].sName;
				fbAlarm[i].CreateEx(TC_Events.AlarmSystem.B1, FALSE, fbSourceInfo);
			B2:
				fbSourceInfo.Clear();
				fbSourceInfo.sName := arrAlarms[i].sName;
				fbAlarm[i].CreateEx(TC_Events.AlarmSystem.B2, FALSE, fbSourceInfo);
			B3:
				fbSourceInfo.Clear();
				fbSourceInfo.sName := arrAlarms[i].sName;
				fbAlarm[i].CreateEx(TC_Events.AlarmSystem.B3, FALSE, fbSourceInfo);
			B4:
				fbSourceInfo.Clear();
				fbSourceInfo.sName := arrAlarms[i].sName;
				fbAlarm[i].CreateEx(TC_Events.AlarmSystem.B4, FALSE, fbSourceInfo);
			B5:
				fbSourceInfo.Clear();
				fbSourceInfo.sName := arrAlarms[i].sName;
				fbAlarm[i].CreateEx(TC_Events.AlarmSystem.B5, FALSE, fbSourceInfo);
			B6:
				fbSourceInfo.Clear();
				fbSourceInfo.sName := arrAlarms[i].sName;
				fbAlarm[i].CreateEx(TC_Events.AlarmSystem.B6, FALSE, fbSourceInfo);
			B7:
				fbSourceInfo.Clear();
				fbSourceInfo.sName := arrAlarms[i].sName;
				fbAlarm[i].CreateEx(TC_Events.AlarmSystem.B7, FALSE, fbSourceInfo);
			B8:
				fbSourceInfo.Clear();
				fbSourceInfo.sName := arrAlarms[i].sName;
				fbAlarm[i].CreateEx(TC_Events.AlarmSystem.B8, FALSE, fbSourceInfo);
			B9:
				fbSourceInfo.Clear();
				fbSourceInfo.sName := arrAlarms[i].sName;
				fbAlarm[i].CreateEx(TC_Events.AlarmSystem.B9, FALSE, fbSourceInfo);
			B10:
				fbSourceInfo.Clear();
				fbSourceInfo.sName := arrAlarms[i].sName;
				fbAlarm[i].CreateEx(TC_Events.AlarmSystem.B10, FALSE, fbSourceInfo);
			B11:
				fbSourceInfo.Clear();
				fbSourceInfo.sName := arrAlarms[i].sName;
				fbAlarm[i].CreateEx(TC_Events.AlarmSystem.B11, FALSE, fbSourceInfo);
			B12:
				fbSourceInfo.Clear();
				fbSourceInfo.sName := arrAlarms[i].sName;
				fbAlarm[i].CreateEx(TC_Events.AlarmSystem.B12, FALSE, fbSourceInfo);
			B13:
				fbSourceInfo.Clear();
				fbSourceInfo.sName := arrAlarms[i].sName;
				fbAlarm[i].CreateEx(TC_Events.AlarmSystem.B13, FALSE, fbSourceInfo);
			B14:
				fbSourceInfo.Clear();
				fbSourceInfo.sName := arrAlarms[i].sName;
				fbAlarm[i].CreateEx(TC_Events.AlarmSystem.B14, FALSE, fbSourceInfo);
			B15:
				fbSourceInfo.Clear();
				fbSourceInfo.sName := arrAlarms[i].sName;
				fbAlarm[i].CreateEx(TC_Events.AlarmSystem.B15, FALSE, fbSourceInfo);
			B16:
				fbSourceInfo.Clear();
				fbSourceInfo.sName := arrAlarms[i].sName;
				fbAlarm[i].CreateEx(TC_Events.AlarmSystem.B16, FALSE, fbSourceInfo);
			B17:
				fbSourceInfo.Clear();
				fbSourceInfo.sName := arrAlarms[i].sName;
				fbAlarm[i].CreateEx(TC_Events.AlarmSystem.B17, FALSE, fbSourceInfo);
			B18:
				fbSourceInfo.Clear();
				fbSourceInfo.sName := arrAlarms[i].sName;
				fbAlarm[i].CreateEx(TC_Events.AlarmSystem.B18, FALSE, fbSourceInfo);
			B20:
				fbSourceInfo.Clear();
				fbSourceInfo.sName := arrAlarms[i].sName;
				fbAlarm[i].CreateEx(TC_Events.AlarmSystem.B20, FALSE, fbSourceInfo);
			B25:
				fbSourceInfo.Clear();
				fbSourceInfo.sName := arrAlarms[i].sName;
				fbAlarm[i].CreateEx(TC_Events.AlarmSystem.B25, FALSE, fbSourceInfo);
			B30:
				fbSourceInfo.Clear();
				fbSourceInfo.sName := arrAlarms[i].sName;
				fbAlarm[i].CreateEx(TC_Events.AlarmSystem.B30, FALSE, fbSourceInfo);
			B40:
				fbSourceInfo.Clear();
				fbSourceInfo.sName := arrAlarms[i].sName;
				fbAlarm[i].CreateEx(TC_Events.AlarmSystem.B40, FALSE, fbSourceInfo);
			B99:
				fbSourceInfo.Clear();
				fbSourceInfo.sName := arrAlarms[i].sName;
				fbAlarm[i].CreateEx(TC_Events.AlarmSystem.B99, FALSE, fbSourceInfo);
			B100:
				fbSourceInfo.Clear();
				fbSourceInfo.sName := arrAlarms[i].sName;
				fbAlarm[i].CreateEx(TC_Events.AlarmSystem.B100, FALSE, fbSourceInfo);
			
		END_CASE
	END_FOR
	
 IF i>=222 THEN
	 bInit:=1;
 END_IF
END_IF
END_ACTION

ACTION RaiseAlarms:
// COMMAND ALARMS BASED ON THE .B OF THE WIN WIND ALARM STUCTURE
    //bRaiseAlarm[1] := FALSE;
	IF arrAlarms[index2].b THEN
   		fbAlarm[index2].ipArguments.Clear().AddString(arrAlarms[index2].Comment);
    	fbAlarm[index2].Raise(0);
	END_IF
END_ACTION

END_PROGRAM

// ---- Alarm System/POUs/02_Alarm_Handling/FB_StatusCodeLogger.TcPOU
FUNCTION_BLOCK FB_StatusCodeLogger
(**********************************************************************************)
(**********************************************************************************)
(*  	VERSION:				001.007

  	PROGRAMMED BY:		Puja
  	Changed BY:				Hardy Patommel
	DATE:					2009-01-21
*)							               				 			
(*-------------------------------------------------------------------------------------------------------*)
 (*  	REVISIONS:
   	Date		|	Version/Author 		|	Remark
	----------------------------------------------------------------------------------------------------
	25-06-2007	|	001.001     HP			|	modified error handling
 	2009-10-26	|	003.001 RM			|	Prepared for Library
		                									 
*)
(*--------------------------------------------------------------------------------------------------------*)
(*  	DESCRIPTION:
	The size of  strings must correspond with the event - structure length in the ring buffer
	memory
	Function block------			
	- sTimeStamp[24]			
	- sKeyAndText[23]			sTrigEventText[80]	>> uiKeyAndTextLen; uiTextLen (*max using length is [uiKeyAndTextLen - sKeySize]*)
	- sUserName[23]			sUserName[24]
	- sBrakeProgram[4]

	Ring buffer-----------
	TYPE ST_LoggedEvent_SC :
	STRUCT
	gtTimeStampUTC	: STRING[23];	(* Time the Statuscode becomes true *)
	gsTrigEvent		: STRING[guiKeyAndTextLen];	(* STRING[91]*)	(*max using length is [uiKeyAndTextLen - sKeySize]*) 
	gsUserName		: STRING[24];	(* name of the user who had the Active Status to do the operation *)
	gsBrakeProgram	: STRING[4];
	Text
*)
(**********************************************************************************)
(**********************************************************************************)
VAR_INPUT
	bTrigEvent				: BOOL;
	sTimeStamp				: STRING[24];
	sTrigEventKey			: STRING[9];					(*sKeySize*)
	sTrigEventText			: STRING[guiKeyAndTextLen]; 	(*max using length is [uiKeyAndTextLen - sKeySize]*)
	sUserName				: STRING[24];
	sBrakeProgram			: STRING[4];
	udNumberOfEventDatas	: UDINT;
	dwArrDataAdr			: ARRAY [1..NUMBER_OF_EVENT_DATAS] OF DWORD;
	udArrDataSize			: ARRAY [1..NUMBER_OF_EVENT_DATAS] OF UDINT;
	eDataType				: ARRAY [1..NUMBER_OF_EVENT_DATAS] OF E_DataType;
	sHeaderOfEventData		: ARRAY [1..giGeneralLoggerChannelInUsed] OF STRING(giGeneralLenghtOfName);
	dwLoggedEventAdr		: DWORD;
	udLoggedEventSize		: UDINT;
	stFileSetup				: ST_FileSetup_SC;
	bWriteDayFile			: BOOL;
	stFileSetupDayFile		: ST_FileSetup_SC;

	CheckLog:		BOOL;
	ResetErrCnt:		BOOL;
END_VAR
VAR_OUTPUT
	bError					: BOOL;
	nErrID					: UDINT;
END_VAR
VAR
	bInitNovRAM				: BOOL := TRUE;
	bInit						: BOOL := TRUE; (*Used for the logger initialisation*)

	sKeyAndText				: STRING[guiKeyAndTextLen];
	udCurrentAddIndex		: UDINT;
	udOldestAddIndex			: UDINT;
	udUsedVal				: UDINT;
	udNumberOfValues		: UDINT;
	udCounter				: INT;
	dwBufferStartAdr 			: DWORD;
	dwBufferEndAdr			: DWORD;
	dwTransferBufferStartAdr 	: DWORD;
	dwTransferBufferEndAdr 	: DWORD;
	udSizeOfeachBlock		: UDINT;
	udOldValuesToBeCopied	: UDINT;
	iNewValues	 			: INT;
	iNumberOfValues			: INT;
	iNumberOfEventDatas		: INT;
	i						: INT;
	bWriteData				: BOOL; (* indicate ready to write *)
	sTab					: STRING[2] := '$T';
	sLineFeed				: STRING[4] := '$R$N';
	iEntriesWritten			: INT;
	iAddOffset				: INT;
	bCheck					: BOOL;
	iIdx						: INT := 1;
	state					: INT;
	fbWriteEventData			: FB_WriteEventData;
	fbWriteEventData_Day		: FB_WriteEventData_Day;
	bWriteDayFileCopy		: BOOL;
	bInitError					: BOOL;
	rTrigErrorWriteData1		: R_TRIG; (*for diagnostic*)
	rTrigErrorWriteData2		: R_TRIG; (*for diagnostic*)
	iErrCounterEventData		: UINT;
	iErrCounterEventData_Day	: UINT;
	ar_iAddOffset				: ARRAY [1..4] OF INT;
	udValuesNotWritten		: UDINT;
	strPathNameTemp		: T_MaxString;
	uiCheckEntryLength		: UINT;		(*for check the length for ring buffer entry size*)
	iSizeOf					: INT;
	uiCheckLenghtError		: UINT;		(*Counter of length error*)
	strLastKeyError			: STRING[guiKeyAndTextLen];
	uiLENsTrigEventText		: UINT;		(*actual length of Statuscode description*)
	uiLENsMaxText			: UINT;
END_VAR
VAR PERSISTENT
	nNextPointerLoc			: DINT; (*next entry line ring buffer Statuscode, persistent declaration for pc system without novram*)
END_VAR

(*========== START OF FUNCTION_BLOCK / PROGRAMM ============*)

	(*==========================================================*)
	(*  				Initialisation (Read from Novram)				       *)
	(*==========================================================*)
(*	IF gbReadFromNovram AND NOT gbRestoreFromNovram_StatuscodeLogger THEN							(*NEEDED?*)
		nNextPointerLoc:= strucFromNOVRAM.iRingBuffer_NextPointerLocation;
		gbRestoreFromNovram_StatuscodeLogger:= TRUE;
		bInitNovRAM:= FALSE;
	ELSIF NOT gbReadFromNovram THEN
		bInitNovRAM:= FALSE;
	END_IF;
	
*)
		bInitNovRAM:= FALSE;																				(*NEEDED? just added; when oben aktiviert, nicht benötigt*)

	(*==========================================================*)
	(*  Counter for diagnostic   *)
	(*==========================================================*)
	IF ResetErrCnt THEN																					(*NEEDED?*)
		iErrCounterEventData 		:= 0;
		iErrCounterEventData_Day 	:= 0;
	END_IF


	CASE state OF
		0:
		(* wait for the entries *)
		fbWriteEventData( bExecute:= FALSE,nNextPointerLoc	:= nNextPointerLoc,);
		IF bWriteData AND NOT bInitNovRAM THEN (* if entries available and sorted *)
			fbWriteEventData(
				bExecute				:= bWriteData,
				sNetId					:= stFileSetup.sNetId,
				sPathName				:= stFileSetup.sPathName,
				dwTransferBufferStartAdr	:= dwTransferBufferStartAdr,
				iNewValues				:= (iIdx-1),
				udNumberofValues		:= udNumberofValues,
				udArrDataSize			:= udArrDataSize,
				udNumberOfEventDatas	:= udNumberOfEventDatas,
				sHeaderOfEventData	:= sHeaderOfEventData,
				iHeaderLEN				:= giRingBufferFileHeaderLEN,
				eDataType				:= eDataType,
				nNextPointerLoc			:= nNextPointerLoc,
				bBusy					=> ,
				bDone					=> ,
				bError					=> bError,
				nErrId					=> nErrId );

			IF bWriteDayFile THEN

				(* Get the right name by initialization and
				   Change the path name by every day for the unlimited event logger file..*)
				(*+++++++++++++++++++++++++++++++++++++++++++++++++++++*)
				IF Lib_strucSystemTime.wDay <> gwNewDayForLogger THEN
					strPathNameTemp :='j'(*  FUN_DateFileNameWithSpace(gsSC_PathName, Lib_strucSystemTime,'')ACTION*) ;
					strPathNameTemp := CONCAT(strPathNameTemp ,'  ');
					fbSCLogger.stFileSetupDayFile.sTotalName :=  CONCAT(strPathNameTemp,fbSCLogger.stFileSetupDayFile.sName);
				END_IF
				gwNewDayForLogger := Lib_strucSystemTime.wDay;

